   // UNI[2929] := 16#94A6;
   // UNI[2930] := 16#4FB5;
   // UNI[2931] := 16#4EB2;
   // UNI[2932] := 16#79E6;
   // UNI[2933] := 16#7434;
   // UNI[2934] := 16#52E4;
   // UNI[2935] := 16#82B9;
   // UNI[2936] := 16#64D2;
   // UNI[2937] := 16#79BD;
   // UNI[2938] := 16#5BDD;
   // UNI[2939] := 16#6C81;
   // UNI[2940] := 16#9752;
   // UNI[2941] := 16#8F7B;
   // UNI[2942] := 16#6C22;
   // UNI[2943] := 16#503E;
   // UNI[2944] := 16#537F;
   // UNI[2945] := 16#6E05;
   // UNI[2946] := 16#64CE;
   // UNI[2947] := 16#6674;
   // UNI[2948] := 16#6C30;
   // UNI[2949] := 16#60C5;
   // UNI[2950] := 16#9877;
   // UNI[2951] := 16#8BF7;
   // UNI[2952] := 16#5E86;
   // UNI[2953] := 16#743C;
   // UNI[2954] := 16#7A77;
   // UNI[2955] := 16#79CB;
   // UNI[2956] := 16#4E18;
   // UNI[2957] := 16#90B1;
   // UNI[2958] := 16#7403;
   // UNI[2959] := 16#6C42;
   // UNI[2960] := 16#56DA;
   // UNI[2961] := 16#914B;
   // UNI[2962] := 16#6CC5;
   // UNI[2963] := 16#8D8B;
   // UNI[2964] := 16#533A;
   // UNI[2965] := 16#86C6;
   // UNI[2966] := 16#66F2;
   // UNI[2967] := 16#8EAF;
   // UNI[2968] := 16#5C48;
   // UNI[2969] := 16#9A71;
   // UNI[2970] := 16#6E20;
   // UNI[2971] := 16#53D6;
   // UNI[2972] := 16#5A36;
   // UNI[2973] := 16#9F8B;
   // UNI[2974] := 16#8DA3;
   // UNI[2975] := 16#53BB;
   // UNI[2976] := 16#5708;
   // UNI[2977] := 16#98A7;
   // UNI[2978] := 16#6743;
   // UNI[2979] := 16#919B;
   // UNI[2980] := 16#6CC9;
   // UNI[2981] := 16#5168;
   // UNI[2982] := 16#75CA;
   // UNI[2983] := 16#62F3;
   // UNI[2984] := 16#72AC;
   // UNI[2985] := 16#5238;
   // UNI[2986] := 16#529D;
   // UNI[2987] := 16#7F3A;
   // UNI[2988] := 16#7094;
   // UNI[2989] := 16#7638;
   // UNI[2990] := 16#5374;
   // UNI[2991] := 16#9E4A;
   // UNI[2992] := 16#69B7;
   // UNI[2993] := 16#786E;
   // UNI[2994] := 16#96C0;
   // UNI[2995] := 16#88D9;
   // UNI[2996] := 16#7FA4;
   // UNI[2997] := 16#7136;
   // UNI[2998] := 16#71C3;
   // UNI[2999] := 16#5189;
   // UNI[3000] := 16#67D3;
   // UNI[3001] := 16#74E4;
   // UNI[3002] := 16#58E4;
   // UNI[3003] := 16#6518;
   // UNI[3004] := 16#56B7;
   // UNI[3005] := 16#8BA9;
   // UNI[3006] := 16#9976;
   // UNI[3007] := 16#6270;
   // UNI[3008] := 16#7ED5;
   // UNI[3009] := 16#60F9;
   // UNI[3010] := 16#70ED;
   // UNI[3011] := 16#58EC;
   // UNI[3012] := 16#4EC1;
   // UNI[3013] := 16#4EBA;
   // UNI[3014] := 16#5FCD;
   // UNI[3015] := 16#97E7;
   // UNI[3016] := 16#4EFB;
   // UNI[3017] := 16#8BA4;
   // UNI[3018] := 16#5203;
   // UNI[3019] := 16#598A;
   // UNI[3020] := 16#7EAB;
   // UNI[3021] := 16#6254;
   // UNI[3022] := 16#4ECD;
   // UNI[3023] := 16#65E5;
   // UNI[3024] := 16#620E;
   // UNI[3025] := 16#8338;
   // UNI[3026] := 16#84C9;
   // UNI[3027] := 16#8363;
   // UNI[3028] := 16#878D;
   // UNI[3029] := 16#7194;
   // UNI[3030] := 16#6EB6;
   // UNI[3031] := 16#5BB9;
   // UNI[3032] := 16#7ED2;
   // UNI[3033] := 16#5197;
   // UNI[3034] := 16#63C9;
   // UNI[3035] := 16#67D4;
   // UNI[3036] := 16#8089;
   // UNI[3037] := 16#8339;
   // UNI[3038] := 16#8815;
   // UNI[3039] := 16#5112;
   // UNI[3040] := 16#5B7A;
   // UNI[3041] := 16#5982;
   // UNI[3042] := 16#8FB1;
   // UNI[3043] := 16#4E73;
   // UNI[3044] := 16#6C5D;
   // UNI[3045] := 16#5165;
   // UNI[3046] := 16#8925;
   // UNI[3047] := 16#8F6F;
   // UNI[3048] := 16#962E;
   // UNI[3049] := 16#854A;
   // UNI[3050] := 16#745E;
   // UNI[3051] := 16#9510;
   // UNI[3052] := 16#95F0;
   // UNI[3053] := 16#6DA6;
   // UNI[3054] := 16#82E5;
   // UNI[3055] := 16#5F31;
   // UNI[3056] := 16#6492;
   // UNI[3057] := 16#6D12;
   // UNI[3058] := 16#8428;
   // UNI[3059] := 16#816E;
   // UNI[3060] := 16#9CC3;
   // UNI[3061] := 16#585E;
   // UNI[3062] := 16#8D5B;
   // UNI[3063] := 16#4E09;
   // UNI[3064] := 16#53C1;
   // UNI[3065] := 16#4F1E;
   // UNI[3066] := 16#6563;
   // UNI[3067] := 16#6851;
   // UNI[3068] := 16#55D3;
   // UNI[3069] := 16#4E27;
   // UNI[3070] := 16#6414;
   // UNI[3071] := 16#9A9A;
   // UNI[3072] := 16#626B;
   // UNI[3073] := 16#5AC2;
   // UNI[3074] := 16#745F;
   // UNI[3075] := 16#8272;
   // UNI[3076] := 16#6DA9;
   // UNI[3077] := 16#68EE;
   // UNI[3078] := 16#50E7;
   // UNI[3079] := 16#838E;
   // UNI[3080] := 16#7802;
   // UNI[3081] := 16#6740;
   // UNI[3082] := 16#5239;
   // UNI[3083] := 16#6C99;
   // UNI[3084] := 16#7EB1;
   // UNI[3085] := 16#50BB;
   // UNI[3086] := 16#5565;
   // UNI[3087] := 16#715E;
   // UNI[3088] := 16#7B5B;
   // UNI[3089] := 16#6652;
   // UNI[3090] := 16#73CA;
   // UNI[3091] := 16#82EB;
   // UNI[3092] := 16#6749;
   // UNI[3093] := 16#5C71;
   // UNI[3094] := 16#5220;
   // UNI[3095] := 16#717D;
   // UNI[3096] := 16#886B;
   // UNI[3097] := 16#95EA;
   // UNI[3098] := 16#9655;
   // UNI[3099] := 16#64C5;
   // UNI[3100] := 16#8D61;
   // UNI[3101] := 16#81B3;
   // UNI[3102] := 16#5584;
   // UNI[3103] := 16#6C55;
   // UNI[3104] := 16#6247;
   // UNI[3105] := 16#7F2E;
   // UNI[3106] := 16#5892;
   // UNI[3107] := 16#4F24;
   // UNI[3108] := 16#5546;
   // UNI[3109] := 16#8D4F;
   // UNI[3110] := 16#664C;
   // UNI[3111] := 16#4E0A;
   // UNI[3112] := 16#5C1A;
   // UNI[3113] := 16#88F3;
   // UNI[3114] := 16#68A2;
   // UNI[3115] := 16#634E;
   // UNI[3116] := 16#7A0D;
   // UNI[3117] := 16#70E7;
   // UNI[3118] := 16#828D;
   // UNI[3119] := 16#52FA;
   // UNI[3120] := 16#97F6;
   // UNI[3121] := 16#5C11;
   // UNI[3122] := 16#54E8;
   // UNI[3123] := 16#90B5;
   // UNI[3124] := 16#7ECD;
   // UNI[3125] := 16#5962;
   // UNI[3126] := 16#8D4A;
   // UNI[3127] := 16#86C7;
   // UNI[3128] := 16#820C;
   // UNI[3129] := 16#820D;
   // UNI[3130] := 16#8D66;
   // UNI[3131] := 16#6444;
   // UNI[3132] := 16#5C04;
   // UNI[3133] := 16#6151;
   // UNI[3134] := 16#6D89;
   // UNI[3135] := 16#793E;
   // UNI[3136] := 16#8BBE;
   // UNI[3137] := 16#7837;
   // UNI[3138] := 16#7533;
   // UNI[3139] := 16#547B;
   // UNI[3140] := 16#4F38;
   // UNI[3141] := 16#8EAB;
   // UNI[3142] := 16#6DF1;
   // UNI[3143] := 16#5A20;
   // UNI[3144] := 16#7EC5;
   // UNI[3145] := 16#795E;
   // UNI[3146] := 16#6C88;
   // UNI[3147] := 16#5BA1;
   // UNI[3148] := 16#5A76;
   // UNI[3149] := 16#751A;
   // UNI[3150] := 16#80BE;
   // UNI[3151] := 16#614E;
   // UNI[3152] := 16#6E17;
   // UNI[3153] := 16#58F0;
   // UNI[3154] := 16#751F;
   // UNI[3155] := 16#7525;
   // UNI[3156] := 16#7272;
   // UNI[3157] := 16#5347;
   // UNI[3158] := 16#7EF3;
   // UNI[3159] := 16#7701;
   // UNI[3160] := 16#76DB;
   // UNI[3161] := 16#5269;
   // UNI[3162] := 16#80DC;
   // UNI[3163] := 16#5723;
   // UNI[3164] := 16#5E08;
   // UNI[3165] := 16#5931;
   // UNI[3166] := 16#72EE;
   // UNI[3167] := 16#65BD;
   // UNI[3168] := 16#6E7F;
   // UNI[3169] := 16#8BD7;
   // UNI[3170] := 16#5C38;
   // UNI[3171] := 16#8671;
   // UNI[3172] := 16#5341;
   // UNI[3173] := 16#77F3;
   // UNI[3174] := 16#62FE;
   // UNI[3175] := 16#65F6;
   // UNI[3176] := 16#4EC0;
   // UNI[3177] := 16#98DF;
   // UNI[3178] := 16#8680;
   // UNI[3179] := 16#5B9E;
   // UNI[3180] := 16#8BC6;
   // UNI[3181] := 16#53F2;
   // UNI[3182] := 16#77E2;
   // UNI[3183] := 16#4F7F;
   // UNI[3184] := 16#5C4E;
   // UNI[3185] := 16#9A76;
   // UNI[3186] := 16#59CB;
   // UNI[3187] := 16#5F0F;
   // UNI[3188] := 16#793A;
   // UNI[3189] := 16#58EB;
   // UNI[3190] := 16#4E16;
   // UNI[3191] := 16#67FF;
   // UNI[3192] := 16#4E8B;
   // UNI[3193] := 16#62ED;
   // UNI[3194] := 16#8A93;
   // UNI[3195] := 16#901D;
   // UNI[3196] := 16#52BF;
   // UNI[3197] := 16#662F;
   // UNI[3198] := 16#55DC;
   // UNI[3199] := 16#566C;
   // UNI[3200] := 16#9002;
   // UNI[3201] := 16#4ED5;
   // UNI[3202] := 16#4F8D;
   // UNI[3203] := 16#91CA;
   // UNI[3204] := 16#9970;
   // UNI[3205] := 16#6C0F;
   // UNI[3206] := 16#5E02;
   // UNI[3207] := 16#6043;
   // UNI[3208] := 16#5BA4;
   // UNI[3209] := 16#89C6;
   // UNI[3210] := 16#8BD5;
   // UNI[3211] := 16#6536;
   // UNI[3212] := 16#624B;
   // UNI[3213] := 16#9996;
   // UNI[3214] := 16#5B88;
   // UNI[3215] := 16#5BFF;
   // UNI[3216] := 16#6388;
   // UNI[3217] := 16#552E;
   // UNI[3218] := 16#53D7;
   // UNI[3219] := 16#7626;
   // UNI[3220] := 16#517D;
   // UNI[3221] := 16#852C;
   // UNI[3222] := 16#67A2;
   // UNI[3223] := 16#68B3;
   // UNI[3224] := 16#6B8A;
   // UNI[3225] := 16#6292;
   // UNI[3226] := 16#8F93;
   // UNI[3227] := 16#53D4;
   // UNI[3228] := 16#8212;
   // UNI[3229] := 16#6DD1;
   // UNI[3230] := 16#758F;
   // UNI[3231] := 16#4E66;
   // UNI[3232] := 16#8D4E;
   // UNI[3233] := 16#5B70;
   // UNI[3234] := 16#719F;
   // UNI[3235] := 16#85AF;
   // UNI[3236] := 16#6691;
   // UNI[3237] := 16#66D9;
   // UNI[3238] := 16#7F72;
   // UNI[3239] := 16#8700;
   // UNI[3240] := 16#9ECD;
   // UNI[3241] := 16#9F20;
   // UNI[3242] := 16#5C5E;
   // UNI[3243] := 16#672F;
   // UNI[3244] := 16#8FF0;
   // UNI[3245] := 16#6811;
   // UNI[3246] := 16#675F;
   // UNI[3247] := 16#620D;
   // UNI[3248] := 16#7AD6;
   // UNI[3249] := 16#5885;
   // UNI[3250] := 16#5EB6;
   // UNI[3251] := 16#6570;
   // UNI[3252] := 16#6F31;
   // UNI[3253] := 16#6055;
   // UNI[3254] := 16#5237;
   // UNI[3255] := 16#800D;
   // UNI[3256] := 16#6454;
   // UNI[3257] := 16#8870;
   // UNI[3258] := 16#7529;
   // UNI[3259] := 16#5E05;
   // UNI[3260] := 16#6813;
   // UNI[3261] := 16#62F4;
   // UNI[3262] := 16#971C;
   // UNI[3263] := 16#53CC;
   // UNI[3264] := 16#723D;
   // UNI[3265] := 16#8C01;
   // UNI[3266] := 16#6C34;
   // UNI[3267] := 16#7761;
   // UNI[3268] := 16#7A0E;
   // UNI[3269] := 16#542E;
   // UNI[3270] := 16#77AC;
   // UNI[3271] := 16#987A;
   // UNI[3272] := 16#821C;
   // UNI[3273] := 16#8BF4;
   // UNI[3274] := 16#7855;
   // UNI[3275] := 16#6714;
   // UNI[3276] := 16#70C1;
   // UNI[3277] := 16#65AF;
   // UNI[3278] := 16#6495;
   // UNI[3279] := 16#5636;
   // UNI[3280] := 16#601D;
   // UNI[3281] := 16#79C1;
   // UNI[3282] := 16#53F8;
   // UNI[3283] := 16#4E1D;
   // UNI[3284] := 16#6B7B;
   // UNI[3285] := 16#8086;
   // UNI[3286] := 16#5BFA;
   // UNI[3287] := 16#55E3;
   // UNI[3288] := 16#56DB;
   // UNI[3289] := 16#4F3A;
   // UNI[3290] := 16#4F3C;
   // UNI[3291] := 16#9972;
   // UNI[3292] := 16#5DF3;
   // UNI[3293] := 16#677E;
   // UNI[3294] := 16#8038;
   // UNI[3295] := 16#6002;
   // UNI[3296] := 16#9882;
   // UNI[3297] := 16#9001;
   // UNI[3298] := 16#5B8B;
   // UNI[3299] := 16#8BBC;
   // UNI[3300] := 16#8BF5;
   // UNI[3301] := 16#641C;
   // UNI[3302] := 16#8258;
   // UNI[3303] := 16#64DE;
   // UNI[3304] := 16#55FD;
   // UNI[3305] := 16#82CF;
   // UNI[3306] := 16#9165;
   // UNI[3307] := 16#4FD7;
   // UNI[3308] := 16#7D20;
   // UNI[3309] := 16#901F;
   // UNI[3310] := 16#7C9F;
   // UNI[3311] := 16#50F3;
   // UNI[3312] := 16#5851;
   // UNI[3313] := 16#6EAF;
   // UNI[3314] := 16#5BBF;
   // UNI[3315] := 16#8BC9;
   // UNI[3316] := 16#8083;
   // UNI[3317] := 16#9178;
   // UNI[3318] := 16#849C;
   // UNI[3319] := 16#7B97;
   // UNI[3320] := 16#867D;
   // UNI[3321] := 16#968B;
   // UNI[3322] := 16#968F;
   // UNI[3323] := 16#7EE5;
   // UNI[3324] := 16#9AD3;
   // UNI[3325] := 16#788E;
   // UNI[3326] := 16#5C81;
   // UNI[3327] := 16#7A57;
   // UNI[3328] := 16#9042;
   // UNI[3329] := 16#96A7;
   // UNI[3330] := 16#795F;
   // UNI[3331] := 16#5B59;
   // UNI[3332] := 16#635F;
   // UNI[3333] := 16#7B0B;
   // UNI[3334] := 16#84D1;
   // UNI[3335] := 16#68AD;
   // UNI[3336] := 16#5506;
   // UNI[3337] := 16#7F29;
   // UNI[3338] := 16#7410;
   // UNI[3339] := 16#7D22;
   // UNI[3340] := 16#9501;
   // UNI[3341] := 16#6240;
   // UNI[3342] := 16#584C;
   // UNI[3343] := 16#4ED6;
   // UNI[3344] := 16#5B83;
   // UNI[3345] := 16#5979;
   // UNI[3346] := 16#5854;
   // UNI[3347] := 16#736D;
   // UNI[3348] := 16#631E;
   // UNI[3349] := 16#8E4B;
   // UNI[3350] := 16#8E0F;
   // UNI[3351] := 16#80CE;
   // UNI[3352] := 16#82D4;
   // UNI[3353] := 16#62AC;
   // UNI[3354] := 16#53F0;
   // UNI[3355] := 16#6CF0;
   // UNI[3356] := 16#915E;
   // UNI[3357] := 16#592A;
   // UNI[3358] := 16#6001;
   // UNI[3359] := 16#6C70;
   // UNI[3360] := 16#574D;
   // UNI[3361] := 16#644A;
   // UNI[3362] := 16#8D2A;
   // UNI[3363] := 16#762B;
   // UNI[3364] := 16#6EE9;
   // UNI[3365] := 16#575B;
   // UNI[3366] := 16#6A80;
   // UNI[3367] := 16#75F0;
   // UNI[3368] := 16#6F6D;
   // UNI[3369] := 16#8C2D;
   // UNI[3370] := 16#8C08;
   // UNI[3371] := 16#5766;
   // UNI[3372] := 16#6BEF;
   // UNI[3373] := 16#8892;
   // UNI[3374] := 16#78B3;
   // UNI[3375] := 16#63A2;
   // UNI[3376] := 16#53F9;
   // UNI[3377] := 16#70AD;
   // UNI[3378] := 16#6C64;
   // UNI[3379] := 16#5858;
   // UNI[3380] := 16#642A;
   // UNI[3381] := 16#5802;
   // UNI[3382] := 16#68E0;
   // UNI[3383] := 16#819B;
   // UNI[3384] := 16#5510;
   // UNI[3385] := 16#7CD6;
   // UNI[3386] := 16#5018;
   // UNI[3387] := 16#8EBA;
   // UNI[3388] := 16#6DCC;
   // UNI[3389] := 16#8D9F;
   // UNI[3390] := 16#70EB;
   // UNI[3391] := 16#638F;
   // UNI[3392] := 16#6D9B;
   // UNI[3393] := 16#6ED4;
   // UNI[3394] := 16#7EE6;
   // UNI[3395] := 16#8404;
   // UNI[3396] := 16#6843;
   // UNI[3397] := 16#9003;
   // UNI[3398] := 16#6DD8;
   // UNI[3399] := 16#9676;
   // UNI[3400] := 16#8BA8;
   // UNI[3401] := 16#5957;
   // UNI[3402] := 16#7279;
   // UNI[3403] := 16#85E4;
   // UNI[3404] := 16#817E;
   // UNI[3405] := 16#75BC;
   // UNI[3406] := 16#8A8A;
   // UNI[3407] := 16#68AF;
   // UNI[3408] := 16#5254;
   // UNI[3409] := 16#8E22;
   // UNI[3410] := 16#9511;
   // UNI[3411] := 16#63D0;
   // UNI[3412] := 16#9898;
   // UNI[3413] := 16#8E44;
   // UNI[3414] := 16#557C;
   // UNI[3415] := 16#4F53;
   // UNI[3416] := 16#66FF;
   // UNI[3417] := 16#568F;
   // UNI[3418] := 16#60D5;
   // UNI[3419] := 16#6D95;
   // UNI[3420] := 16#5243;
   // UNI[3421] := 16#5C49;
   // UNI[3422] := 16#5929;
   // UNI[3423] := 16#6DFB;
   // UNI[3424] := 16#586B;
   // UNI[3425] := 16#7530;
   // UNI[3426] := 16#751C;
   // UNI[3427] := 16#606C;
   // UNI[3428] := 16#8214;
   // UNI[3429] := 16#8146;
   // UNI[3430] := 16#6311;
   // UNI[3431] := 16#6761;
   // UNI[3432] := 16#8FE2;
   // UNI[3433] := 16#773A;
   // UNI[3434] := 16#8DF3;
   // UNI[3435] := 16#8D34;
   // UNI[3436] := 16#94C1;
   // UNI[3437] := 16#5E16;
   // UNI[3438] := 16#5385;
   // UNI[3439] := 16#542C;
   // UNI[3440] := 16#70C3;
   // UNI[3441] := 16#6C40;
   // UNI[3442] := 16#5EF7;
   // UNI[3443] := 16#505C;
   // UNI[3444] := 16#4EAD;
   // UNI[3445] := 16#5EAD;
   // UNI[3446] := 16#633A;
   // UNI[3447] := 16#8247;
   // UNI[3448] := 16#901A;
   // UNI[3449] := 16#6850;
   // UNI[3450] := 16#916E;
   // UNI[3451] := 16#77B3;
   // UNI[3452] := 16#540C;
   // UNI[3453] := 16#94DC;
   // UNI[3454] := 16#5F64;
   // UNI[3455] := 16#7AE5;
   // UNI[3456] := 16#6876;
   // UNI[3457] := 16#6345;
   // UNI[3458] := 16#7B52;
   // UNI[3459] := 16#7EDF;
   // UNI[3460] := 16#75DB;
   // UNI[3461] := 16#5077;
   // UNI[3462] := 16#6295;
   // UNI[3463] := 16#5934;
   // UNI[3464] := 16#900F;
   // UNI[3465] := 16#51F8;
   // UNI[3466] := 16#79C3;
   // UNI[3467] := 16#7A81;
   // UNI[3468] := 16#56FE;
   // UNI[3469] := 16#5F92;
   // UNI[3470] := 16#9014;
   // UNI[3471] := 16#6D82;
   // UNI[3472] := 16#5C60;
   // UNI[3473] := 16#571F;
   // UNI[3474] := 16#5410;
   // UNI[3475] := 16#5154;
   // UNI[3476] := 16#6E4D;
   // UNI[3477] := 16#56E2;
   // UNI[3478] := 16#63A8;
   // UNI[3479] := 16#9893;
   // UNI[3480] := 16#817F;
   // UNI[3481] := 16#8715;
   // UNI[3482] := 16#892A;
   // UNI[3483] := 16#9000;
   // UNI[3484] := 16#541E;
   // UNI[3485] := 16#5C6F;
   // UNI[3486] := 16#81C0;
   // UNI[3487] := 16#62D6;
   // UNI[3488] := 16#6258;
   // UNI[3489] := 16#8131;
   // UNI[3490] := 16#9E35;
   // UNI[3491] := 16#9640;
   // UNI[3492] := 16#9A6E;
   // UNI[3493] := 16#9A7C;
   // UNI[3494] := 16#692D;
   // UNI[3495] := 16#59A5;
   // UNI[3496] := 16#62D3;
   // UNI[3497] := 16#553E;
   // UNI[3498] := 16#6316;
   // UNI[3499] := 16#54C7;
   // UNI[3500] := 16#86D9;
   // UNI[3501] := 16#6D3C;
   // UNI[3502] := 16#5A03;
   // UNI[3503] := 16#74E6;
   // UNI[3504] := 16#889C;
   // UNI[3505] := 16#6B6A;
   // UNI[3506] := 16#5916;
   // UNI[3507] := 16#8C4C;
   // UNI[3508] := 16#5F2F;
   // UNI[3509] := 16#6E7E;
   // UNI[3510] := 16#73A9;
   // UNI[3511] := 16#987D;
   // UNI[3512] := 16#4E38;
   // UNI[3513] := 16#70F7;
   // UNI[3514] := 16#5B8C;
   // UNI[3515] := 16#7897;
   // UNI[3516] := 16#633D;
   // UNI[3517] := 16#665A;
   // UNI[3518] := 16#7696;
   // UNI[3519] := 16#60CB;
   // UNI[3520] := 16#5B9B;
   // UNI[3521] := 16#5A49;
   // UNI[3522] := 16#4E07;
   // UNI[3523] := 16#8155;
   // UNI[3524] := 16#6C6A;
   // UNI[3525] := 16#738B;
   // UNI[3526] := 16#4EA1;
   // UNI[3527] := 16#6789;
   // UNI[3528] := 16#7F51;
   // UNI[3529] := 16#5F80;
   // UNI[3530] := 16#65FA;
   // UNI[3531] := 16#671B;
   // UNI[3532] := 16#5FD8;
   // UNI[3533] := 16#5984;
   // UNI[3534] := 16#5A01;
   // UNI[3535] := 16#5DCD;
   // UNI[3536] := 16#5FAE;
   // UNI[3537] := 16#5371;
   // UNI[3538] := 16#97E6;
   // UNI[3539] := 16#8FDD;
   // UNI[3540] := 16#6845;
   // UNI[3541] := 16#56F4;
   // UNI[3542] := 16#552F;
   // UNI[3543] := 16#60DF;
   // UNI[3544] := 16#4E3A;
   // UNI[3545] := 16#6F4D;
   // UNI[3546] := 16#7EF4;
   // UNI[3547] := 16#82C7;
   // UNI[3548] := 16#840E;
   // UNI[3549] := 16#59D4;
   // UNI[3550] := 16#4F1F;
   // UNI[3551] := 16#4F2A;
   // UNI[3552] := 16#5C3E;
   // UNI[3553] := 16#7EAC;
   // UNI[3554] := 16#672A;
   // UNI[3555] := 16#851A;
   // UNI[3556] := 16#5473;
   // UNI[3557] := 16#754F;
   // UNI[3558] := 16#80C3;
   // UNI[3559] := 16#5582;
   // UNI[3560] := 16#9B4F;
   // UNI[3561] := 16#4F4D;
   // UNI[3562] := 16#6E2D;
   // UNI[3563] := 16#8C13;
   // UNI[3564] := 16#5C09;
   // UNI[3565] := 16#6170;
   // UNI[3566] := 16#536B;
   // UNI[3567] := 16#761F;
   // UNI[3568] := 16#6E29;
   // UNI[3569] := 16#868A;
   // UNI[3570] := 16#6587;
   // UNI[3571] := 16#95FB;
   // UNI[3572] := 16#7EB9;
   // UNI[3573] := 16#543B;
   // UNI[3574] := 16#7A33;
   // UNI[3575] := 16#7D0A;
   // UNI[3576] := 16#95EE;
   // UNI[3577] := 16#55E1;
   // UNI[3578] := 16#7FC1;
   // UNI[3579] := 16#74EE;
   // UNI[3580] := 16#631D;
   // UNI[3581] := 16#8717;
   // UNI[3582] := 16#6DA1;
   // UNI[3583] := 16#7A9D;
   // UNI[3584] := 16#6211;
   // UNI[3585] := 16#65A1;
   // UNI[3586] := 16#5367;
   // UNI[3587] := 16#63E1;
   // UNI[3588] := 16#6C83;
   // UNI[3589] := 16#5DEB;
   // UNI[3590] := 16#545C;
   // UNI[3591] := 16#94A8;
   // UNI[3592] := 16#4E4C;
   // UNI[3593] := 16#6C61;
   // UNI[3594] := 16#8BEC;
   // UNI[3595] := 16#5C4B;
   // UNI[3596] := 16#65E0;
   // UNI[3597] := 16#829C;
   // UNI[3598] := 16#68A7;
   // UNI[3599] := 16#543E;
   // UNI[3600] := 16#5434;
   // UNI[3601] := 16#6BCB;
   // UNI[3602] := 16#6B66;
   // UNI[3603] := 16#4E94;
   // UNI[3604] := 16#6342;
   // UNI[3605] := 16#5348;
   // UNI[3606] := 16#821E;
   // UNI[3607] := 16#4F0D;
   // UNI[3608] := 16#4FAE;
   // UNI[3609] := 16#575E;
   // UNI[3610] := 16#620A;
   // UNI[3611] := 16#96FE;
   // UNI[3612] := 16#6664;
   // UNI[3613] := 16#7269;
   // UNI[3614] := 16#52FF;
   // UNI[3615] := 16#52A1;
   // UNI[3616] := 16#609F;
   // UNI[3617] := 16#8BEF;
   // UNI[3618] := 16#6614;
   // UNI[3619] := 16#7199;
   // UNI[3620] := 16#6790;
   // UNI[3621] := 16#897F;
   // UNI[3622] := 16#7852;
   // UNI[3623] := 16#77FD;
   // UNI[3624] := 16#6670;
   // UNI[3625] := 16#563B;
   // UNI[3626] := 16#5438;
   // UNI[3627] := 16#9521;
   // UNI[3628] := 16#727A;
   // UNI[3629] := 16#7A00;
   // UNI[3630] := 16#606F;
   // UNI[3631] := 16#5E0C;
   // UNI[3632] := 16#6089;
   // UNI[3633] := 16#819D;
   // UNI[3634] := 16#5915;
   // UNI[3635] := 16#60DC;
   // UNI[3636] := 16#7184;
   // UNI[3637] := 16#70EF;
   // UNI[3638] := 16#6EAA;
   // UNI[3639] := 16#6C50;
   // UNI[3640] := 16#7280;
   // UNI[3641] := 16#6A84;
   // UNI[3642] := 16#88AD;
   // UNI[3643] := 16#5E2D;
   // UNI[3644] := 16#4E60;
   // UNI[3645] := 16#5AB3;
   // UNI[3646] := 16#559C;
   // UNI[3647] := 16#94E3;
   // UNI[3648] := 16#6D17;
   // UNI[3649] := 16#7CFB;
   // UNI[3650] := 16#9699;
   // UNI[3651] := 16#620F;
   // UNI[3652] := 16#7EC6;
   // UNI[3653] := 16#778E;
   // UNI[3654] := 16#867E;
   // UNI[3655] := 16#5323;
   // UNI[3656] := 16#971E;
   // UNI[3657] := 16#8F96;
   // UNI[3658] := 16#6687;
   // UNI[3659] := 16#5CE1;
   // UNI[3660] := 16#4FA0;
   // UNI[3661] := 16#72ED;
   // UNI[3662] := 16#4E0B;
   // UNI[3663] := 16#53A6;
   // UNI[3664] := 16#590F;
   // UNI[3665] := 16#5413;
   // UNI[3666] := 16#6380;
   // UNI[3667] := 16#9528;
   // UNI[3668] := 16#5148;
   // UNI[3669] := 16#4ED9;
   // UNI[3670] := 16#9C9C;
   // UNI[3671] := 16#7EA4;
   // UNI[3672] := 16#54B8;
   // UNI[3673] := 16#8D24;
   // UNI[3674] := 16#8854;
   // UNI[3675] := 16#8237;
   // UNI[3676] := 16#95F2;
   // UNI[3677] := 16#6D8E;
   // UNI[3678] := 16#5F26;
   // UNI[3679] := 16#5ACC;
   // UNI[3680] := 16#663E;
   // UNI[3681] := 16#9669;
   // UNI[3682] := 16#73B0;
   // UNI[3683] := 16#732E;
   // UNI[3684] := 16#53BF;
   // UNI[3685] := 16#817A;
   // UNI[3686] := 16#9985;
   // UNI[3687] := 16#7FA1;
   // UNI[3688] := 16#5BAA;
   // UNI[3689] := 16#9677;
   // UNI[3690] := 16#9650;
   // UNI[3691] := 16#7EBF;
   // UNI[3692] := 16#76F8;
   // UNI[3693] := 16#53A2;
   // UNI[3694] := 16#9576;
   // UNI[3695] := 16#9999;
   // UNI[3696] := 16#7BB1;
   // UNI[3697] := 16#8944;
   // UNI[3698] := 16#6E58;
   // UNI[3699] := 16#4E61;
   // UNI[3700] := 16#7FD4;
   // UNI[3701] := 16#7965;
   // UNI[3702] := 16#8BE6;
   // UNI[3703] := 16#60F3;
   // UNI[3704] := 16#54CD;
   // UNI[3705] := 16#4EAB;
   // UNI[3706] := 16#9879;
   // UNI[3707] := 16#5DF7;
   // UNI[3708] := 16#6A61;
   // UNI[3709] := 16#50CF;
   // UNI[3710] := 16#5411;
   // UNI[3711] := 16#8C61;
   // UNI[3712] := 16#8427;
   // UNI[3713] := 16#785D;
   // UNI[3714] := 16#9704;
   // UNI[3715] := 16#524A;
   // UNI[3716] := 16#54EE;
   // UNI[3717] := 16#56A3;
   // UNI[3718] := 16#9500;
   // UNI[3719] := 16#6D88;
   // UNI[3720] := 16#5BB5;
   // UNI[3721] := 16#6DC6;
   // UNI[3722] := 16#6653;
   // UNI[3723] := 16#5C0F;
   // UNI[3724] := 16#5B5D;
   // UNI[3725] := 16#6821;
   // UNI[3726] := 16#8096;
   // UNI[3727] := 16#5578;
   // UNI[3728] := 16#7B11;
   // UNI[3729] := 16#6548;
   // UNI[3730] := 16#6954;
   // UNI[3731] := 16#4E9B;
   // UNI[3732] := 16#6B47;
   // UNI[3733] := 16#874E;
   // UNI[3734] := 16#978B;
   // UNI[3735] := 16#534F;
   // UNI[3736] := 16#631F;
   // UNI[3737] := 16#643A;
   // UNI[3738] := 16#90AA;
   // UNI[3739] := 16#659C;
   // UNI[3740] := 16#80C1;
   // UNI[3741] := 16#8C10;
   // UNI[3742] := 16#5199;
   // UNI[3743] := 16#68B0;
   // UNI[3744] := 16#5378;
   // UNI[3745] := 16#87F9;
   // UNI[3746] := 16#61C8;
   // UNI[3747] := 16#6CC4;
   // UNI[3748] := 16#6CFB;
   // UNI[3749] := 16#8C22;
   // UNI[3750] := 16#5C51;
   // UNI[3751] := 16#85AA;
   // UNI[3752] := 16#82AF;
   // UNI[3753] := 16#950C;
   // UNI[3754] := 16#6B23;
   // UNI[3755] := 16#8F9B;
   // UNI[3756] := 16#65B0;
   // UNI[3757] := 16#5FFB;
   // UNI[3758] := 16#5FC3;
   // UNI[3759] := 16#4FE1;
   // UNI[3760] := 16#8845;
   // UNI[3761] := 16#661F;
   // UNI[3762] := 16#8165;
   // UNI[3763] := 16#7329;
   // UNI[3764] := 16#60FA;
   // UNI[3765] := 16#5174;
   // UNI[3766] := 16#5211;
   // UNI[3767] := 16#578B;
   // UNI[3768] := 16#5F62;
   // UNI[3769] := 16#90A2;
   // UNI[3770] := 16#884C;
   // UNI[3771] := 16#9192;
   // UNI[3772] := 16#5E78;
   // UNI[3773] := 16#674F;
   // UNI[3774] := 16#6027;
   // UNI[3775] := 16#59D3;
   // UNI[3776] := 16#5144;
   // UNI[3777] := 16#51F6;
   // UNI[3778] := 16#80F8;
   // UNI[3779] := 16#5308;
   // UNI[3780] := 16#6C79;
   // UNI[3781] := 16#96C4;
   // UNI[3782] := 16#718A;
   // UNI[3783] := 16#4F11;
   // UNI[3784] := 16#4FEE;
   // UNI[3785] := 16#7F9E;
   // UNI[3786] := 16#673D;
   // UNI[3787] := 16#55C5;
   // UNI[3788] := 16#9508;
   // UNI[3789] := 16#79C0;
   // UNI[3790] := 16#8896;
   // UNI[3791] := 16#7EE3;
   // UNI[3792] := 16#589F;
   // UNI[3793] := 16#620C;
   // UNI[3794] := 16#9700;
   // UNI[3795] := 16#865A;
   // UNI[3796] := 16#5618;
   // UNI[3797] := 16#987B;
   // UNI[3798] := 16#5F90;
   // UNI[3799] := 16#8BB8;
   // UNI[3800] := 16#84C4;
   // UNI[3801] := 16#9157;
   // UNI[3802] := 16#53D9;
   // UNI[3803] := 16#65ED;
   // UNI[3804] := 16#5E8F;
   // UNI[3805] := 16#755C;
   // UNI[3806] := 16#6064;
   // UNI[3807] := 16#7D6E;
   // UNI[3808] := 16#5A7F;
   // UNI[3809] := 16#7EEA;
   // UNI[3810] := 16#7EED;
   // UNI[3811] := 16#8F69;
   // UNI[3812] := 16#55A7;
   // UNI[3813] := 16#5BA3;
   // UNI[3814] := 16#60AC;
   // UNI[3815] := 16#65CB;
   // UNI[3816] := 16#7384;
   // UNI[3817] := 16#9009;
   // UNI[3818] := 16#7663;
   // UNI[3819] := 16#7729;
   // UNI[3820] := 16#7EDA;
   // UNI[3821] := 16#9774;
   // UNI[3822] := 16#859B;
   // UNI[3823] := 16#5B66;
   // UNI[3824] := 16#7A74;
   // UNI[3825] := 16#96EA;
   // UNI[3826] := 16#8840;
   // UNI[3827] := 16#52CB;
   // UNI[3828] := 16#718F;
   // UNI[3829] := 16#5FAA;
   // UNI[3830] := 16#65EC;
   // UNI[3831] := 16#8BE2;
   // UNI[3832] := 16#5BFB;
   // UNI[3833] := 16#9A6F;
   // UNI[3834] := 16#5DE1;
   // UNI[3835] := 16#6B89;
   // UNI[3836] := 16#6C5B;
   // UNI[3837] := 16#8BAD;
   // UNI[3838] := 16#8BAF;
   // UNI[3839] := 16#900A;
   // UNI[3840] := 16#8FC5;
   // UNI[3841] := 16#538B;
   // UNI[3842] := 16#62BC;
   // UNI[3843] := 16#9E26;
   // UNI[3844] := 16#9E2D;
   // UNI[3845] := 16#5440;
   // UNI[3846] := 16#4E2B;
   // UNI[3847] := 16#82BD;
   // UNI[3848] := 16#7259;
   // UNI[3849] := 16#869C;
   // UNI[3850] := 16#5D16;
   // UNI[3851] := 16#8859;
   // UNI[3852] := 16#6DAF;
   // UNI[3853] := 16#96C5;
   // UNI[3854] := 16#54D1;
   // UNI[3855] := 16#4E9A;
   // UNI[3856] := 16#8BB6;
   // UNI[3857] := 16#7109;
   // UNI[3858] := 16#54BD;
   // UNI[3859] := 16#9609;
   // UNI[3860] := 16#70DF;
   // UNI[3861] := 16#6DF9;
   // UNI[3862] := 16#76D0;
   // UNI[3863] := 16#4E25;
   // UNI[3864] := 16#7814;
   // UNI[3865] := 16#8712;
   // UNI[3866] := 16#5CA9;
   // UNI[3867] := 16#5EF6;
   // UNI[3868] := 16#8A00;
   // UNI[3869] := 16#989C;
   // UNI[3870] := 16#960E;
   // UNI[3871] := 16#708E;
   // UNI[3872] := 16#6CBF;
   // UNI[3873] := 16#5944;
   // UNI[3874] := 16#63A9;
   // UNI[3875] := 16#773C;
   // UNI[3876] := 16#884D;
   // UNI[3877] := 16#6F14;
   // UNI[3878] := 16#8273;
   // UNI[3879] := 16#5830;
   // UNI[3880] := 16#71D5;
   // UNI[3881] := 16#538C;
   // UNI[3882] := 16#781A;
   // UNI[3883] := 16#96C1;
   // UNI[3884] := 16#5501;
   // UNI[3885] := 16#5F66;
   // UNI[3886] := 16#7130;
   // UNI[3887] := 16#5BB4;
   // UNI[3888] := 16#8C1A;
   // UNI[3889] := 16#9A8C;
   // UNI[3890] := 16#6B83;
   // UNI[3891] := 16#592E;
   // UNI[3892] := 16#9E2F;
   // UNI[3893] := 16#79E7;
   // UNI[3894] := 16#6768;
   // UNI[3895] := 16#626C;
   // UNI[3896] := 16#4F6F;
   // UNI[3897] := 16#75A1;
   // UNI[3898] := 16#7F8A;
   // UNI[3899] := 16#6D0B;
   // UNI[3900] := 16#9633;
   // UNI[3901] := 16#6C27;
   // UNI[3902] := 16#4EF0;
   // UNI[3903] := 16#75D2;
   // UNI[3904] := 16#517B;
   // UNI[3905] := 16#6837;
   // UNI[3906] := 16#6F3E;
   // UNI[3907] := 16#9080;
   // UNI[3908] := 16#8170;
   // UNI[3909] := 16#5996;
   // UNI[3910] := 16#7476;
   // UNI[3911] := 16#6447;
   // UNI[3912] := 16#5C27;
   // UNI[3913] := 16#9065;
   // UNI[3914] := 16#7A91;
   // UNI[3915] := 16#8C23;
   // UNI[3916] := 16#59DA;
   // UNI[3917] := 16#54AC;
   // UNI[3918] := 16#8200;
   // UNI[3919] := 16#836F;
   // UNI[3920] := 16#8981;
   // UNI[3921] := 16#8000;
   // UNI[3922] := 16#6930;
   // UNI[3923] := 16#564E;
   // UNI[3924] := 16#8036;
   // UNI[3925] := 16#7237;
   // UNI[3926] := 16#91CE;
   // UNI[3927] := 16#51B6;
   // UNI[3928] := 16#4E5F;
   // UNI[3929] := 16#9875;
   // UNI[3930] := 16#6396;
   // UNI[3931] := 16#4E1A;
   // UNI[3932] := 16#53F6;
   // UNI[3933] := 16#66F3;
   // UNI[3934] := 16#814B;
   // UNI[3935] := 16#591C;
   // UNI[3936] := 16#6DB2;
   // UNI[3937] := 16#4E00;
   // UNI[3938] := 16#58F9;
   // UNI[3939] := 16#533B;
   // UNI[3940] := 16#63D6;
   // UNI[3941] := 16#94F1;
   // UNI[3942] := 16#4F9D;
   // UNI[3943] := 16#4F0A;
   // UNI[3944] := 16#8863;
   // UNI[3945] := 16#9890;
   // UNI[3946] := 16#5937;
   // UNI[3947] := 16#9057;
   // UNI[3948] := 16#79FB;
   // UNI[3949] := 16#4EEA;
   // UNI[3950] := 16#80F0;
   // UNI[3951] := 16#7591;
   // UNI[3952] := 16#6C82;
   // UNI[3953] := 16#5B9C;
   // UNI[3954] := 16#59E8;
   // UNI[3955] := 16#5F5D;
   // UNI[3956] := 16#6905;
   // UNI[3957] := 16#8681;
   // UNI[3958] := 16#501A;
   // UNI[3959] := 16#5DF2;
   // UNI[3960] := 16#4E59;
   // UNI[3961] := 16#77E3;
   // UNI[3962] := 16#4EE5;
   // UNI[3963] := 16#827A;
   // UNI[3964] := 16#6291;
   // UNI[3965] := 16#6613;
   // UNI[3966] := 16#9091;
   // UNI[3967] := 16#5C79;
   // UNI[3968] := 16#4EBF;
   // UNI[3969] := 16#5F79;
   // UNI[3970] := 16#81C6;
   // UNI[3971] := 16#9038;
   // UNI[3972] := 16#8084;
   // UNI[3973] := 16#75AB;
   // UNI[3974] := 16#4EA6;
   // UNI[3975] := 16#88D4;
   // UNI[3976] := 16#610F;
   // UNI[3977] := 16#6BC5;
   // UNI[3978] := 16#5FC6;
   // UNI[3979] := 16#4E49;
   // UNI[3980] := 16#76CA;
   // UNI[3981] := 16#6EA2;
   // UNI[3982] := 16#8BE3;
   // UNI[3983] := 16#8BAE;
   // UNI[3984] := 16#8C0A;
   // UNI[3985] := 16#8BD1;
   // UNI[3986] := 16#5F02;
   // UNI[3987] := 16#7FFC;
   // UNI[3988] := 16#7FCC;
   // UNI[3989] := 16#7ECE;
   // UNI[3990] := 16#8335;
   // UNI[3991] := 16#836B;
   // UNI[3992] := 16#56E0;
   // UNI[3993] := 16#6BB7;
   // UNI[3994] := 16#97F3;
   // UNI[3995] := 16#9634;
   // UNI[3996] := 16#59FB;
   // UNI[3997] := 16#541F;
   // UNI[3998] := 16#94F6;
   // UNI[3999] := 16#6DEB;
   // UNI[4000] := 16#5BC5;
   // UNI[4001] := 16#996E;
   // UNI[4002] := 16#5C39;
   // UNI[4003] := 16#5F15;
   // UNI[4004] := 16#9690;
   // UNI[4005] := 16#5370;
   // UNI[4006] := 16#82F1;
   // UNI[4007] := 16#6A31;
   // UNI[4008] := 16#5A74;
   // UNI[4009] := 16#9E70;
   // UNI[4010] := 16#5E94;
   // UNI[4011] := 16#7F28;
   // UNI[4012] := 16#83B9;
   // UNI[4013] := 16#8424;
   // UNI[4014] := 16#8425;
   // UNI[4015] := 16#8367;
   // UNI[4016] := 16#8747;
   // UNI[4017] := 16#8FCE;
   // UNI[4018] := 16#8D62;
   // UNI[4019] := 16#76C8;
   // UNI[4020] := 16#5F71;
   // UNI[4021] := 16#9896;
   // UNI[4022] := 16#786C;
   // UNI[4023] := 16#6620;
   // UNI[4024] := 16#54DF;
   // UNI[4025] := 16#62E5;
   // UNI[4026] := 16#4F63;
   // UNI[4027] := 16#81C3;
   // UNI[4028] := 16#75C8;
   // UNI[4029] := 16#5EB8;
   // UNI[4030] := 16#96CD;
   // UNI[4031] := 16#8E0A;
   // UNI[4032] := 16#86F9;
   // UNI[4033] := 16#548F;
   // UNI[4034] := 16#6CF3;
   // UNI[4035] := 16#6D8C;
   // UNI[4036] := 16#6C38;
   // UNI[4037] := 16#607F;
   // UNI[4038] := 16#52C7;
   // UNI[4039] := 16#7528;
   // UNI[4040] := 16#5E7D;
   // UNI[4041] := 16#4F18;
   // UNI[4042] := 16#60A0;
   // UNI[4043] := 16#5FE7;
   // UNI[4044] := 16#5C24;
   // UNI[4045] := 16#7531;
   // UNI[4046] := 16#90AE;
   // UNI[4047] := 16#94C0;
   // UNI[4048] := 16#72B9;
   // UNI[4049] := 16#6CB9;
   // UNI[4050] := 16#6E38;
   // UNI[4051] := 16#9149;
   // UNI[4052] := 16#6709;
   // UNI[4053] := 16#53CB;
   // UNI[4054] := 16#53F3;
   // UNI[4055] := 16#4F51;
   // UNI[4056] := 16#91C9;
   // UNI[4057] := 16#8BF1;
   // UNI[4058] := 16#53C8;
   // UNI[4059] := 16#5E7C;
   // UNI[4060] := 16#8FC2;
   // UNI[4061] := 16#6DE4;
   // UNI[4062] := 16#4E8E;
   // UNI[4063] := 16#76C2;
   // UNI[4064] := 16#6986;
   // UNI[4065] := 16#865E;
   // UNI[4066] := 16#611A;
   // UNI[4067] := 16#8206;
   // UNI[4068] := 16#4F59;
   // UNI[4069] := 16#4FDE;
   // UNI[4070] := 16#903E;
   // UNI[4071] := 16#9C7C;
   // UNI[4072] := 16#6109;
   // UNI[4073] := 16#6E1D;
   // UNI[4074] := 16#6E14;
   // UNI[4075] := 16#9685;
   // UNI[4076] := 16#4E88;
   // UNI[4077] := 16#5A31;
   // UNI[4078] := 16#96E8;
   // UNI[4079] := 16#4E0E;
   // UNI[4080] := 16#5C7F;
   // UNI[4081] := 16#79B9;
   // UNI[4082] := 16#5B87;
   // UNI[4083] := 16#8BED;
   // UNI[4084] := 16#7FBD;
   // UNI[4085] := 16#7389;
   // UNI[4086] := 16#57DF;
   // UNI[4087] := 16#828B;
   // UNI[4088] := 16#90C1;
   // UNI[4089] := 16#5401;
   // UNI[4090] := 16#9047;
   // UNI[4091] := 16#55BB;
   // UNI[4092] := 16#5CEA;
   // UNI[4093] := 16#5FA1;
   // UNI[4094] := 16#6108;
   // UNI[4095] := 16#6B32;
   // UNI[4096] := 16#72F1;
   // UNI[4097] := 16#80B2;
   // UNI[4098] := 16#8A89;
   // UNI[4099] := 16#6D74;
   // UNI[4100] := 16#5BD3;
   // UNI[4101] := 16#88D5;
   // UNI[4102] := 16#9884;
   // UNI[4103] := 16#8C6B;
   // UNI[4104] := 16#9A6D;
   // UNI[4105] := 16#9E33;
   // UNI[4106] := 16#6E0A;
   // UNI[4107] := 16#51A4;
   // UNI[4108] := 16#5143;
   // UNI[4109] := 16#57A3;
   // UNI[4110] := 16#8881;
   // UNI[4111] := 16#539F;
   // UNI[4112] := 16#63F4;
   // UNI[4113] := 16#8F95;
   // UNI[4114] := 16#56ED;
   // UNI[4115] := 16#5458;
   // UNI[4116] := 16#5706;
   // UNI[4117] := 16#733F;
   // UNI[4118] := 16#6E90;
   // UNI[4119] := 16#7F18;
   // UNI[4120] := 16#8FDC;
   // UNI[4121] := 16#82D1;
   // UNI[4122] := 16#613F;
   // UNI[4123] := 16#6028;
   // UNI[4124] := 16#9662;
   // UNI[4125] := 16#66F0;
   // UNI[4126] := 16#7EA6;
   // UNI[4127] := 16#8D8A;
   // UNI[4128] := 16#8DC3;
   // UNI[4129] := 16#94A5;
   // UNI[4130] := 16#5CB3;
   // UNI[4131] := 16#7CA4;
   // UNI[4132] := 16#6708;
   // UNI[4133] := 16#60A6;
   // UNI[4134] := 16#9605;
   // UNI[4135] := 16#8018;
   // UNI[4136] := 16#4E91;
   // UNI[4137] := 16#90E7;
   // UNI[4138] := 16#5300;
   // UNI[4139] := 16#9668;
   // UNI[4140] := 16#5141;
   // UNI[4141] := 16#8FD0;
   // UNI[4142] := 16#8574;
   // UNI[4143] := 16#915D;
   // UNI[4144] := 16#6655;
   // UNI[4145] := 16#97F5;
   // UNI[4146] := 16#5B55;
   // UNI[4147] := 16#531D;
   // UNI[4148] := 16#7838;
   // UNI[4149] := 16#6742;
   // UNI[4150] := 16#683D;
   // UNI[4151] := 16#54C9;
   // UNI[4152] := 16#707E;
   // UNI[4153] := 16#5BB0;
   // UNI[4154] := 16#8F7D;
   // UNI[4155] := 16#518D;
   // UNI[4156] := 16#5728;
   // UNI[4157] := 16#54B1;
   // UNI[4158] := 16#6512;
   // UNI[4159] := 16#6682;
   // UNI[4160] := 16#8D5E;
   // UNI[4161] := 16#8D43;
   // UNI[4162] := 16#810F;
   // UNI[4163] := 16#846C;
   // UNI[4164] := 16#906D;
   // UNI[4165] := 16#7CDF;
   // UNI[4166] := 16#51FF;
   // UNI[4167] := 16#85FB;
   // UNI[4168] := 16#67A3;
   // UNI[4169] := 16#65E9;
   // UNI[4170] := 16#6FA1;
   // UNI[4171] := 16#86A4;
   // UNI[4172] := 16#8E81;
   // UNI[4173] := 16#566A;
   // UNI[4174] := 16#9020;
   // UNI[4175] := 16#7682;
   // UNI[4176] := 16#7076;
   // UNI[4177] := 16#71E5;
   // UNI[4178] := 16#8D23;
   // UNI[4179] := 16#62E9;
   // UNI[4180] := 16#5219;
   // UNI[4181] := 16#6CFD;
   // UNI[4182] := 16#8D3C;
   // UNI[4183] := 16#600E;
   // UNI[4184] := 16#589E;
   // UNI[4185] := 16#618E;
   // UNI[4186] := 16#66FE;
   // UNI[4187] := 16#8D60;
   // UNI[4188] := 16#624E;
   // UNI[4189] := 16#55B3;
   // UNI[4190] := 16#6E23;
   // UNI[4191] := 16#672D;
   // UNI[4192] := 16#8F67;
   // UNI[4193] := 16#94E1;
   // UNI[4194] := 16#95F8;
   // UNI[4195] := 16#7728;
   // UNI[4196] := 16#6805;
   // UNI[4197] := 16#69A8;
   // UNI[4198] := 16#548B;
   // UNI[4199] := 16#4E4D;
   // UNI[4200] := 16#70B8;
   // UNI[4201] := 16#8BC8;
   // UNI[4202] := 16#6458;
   // UNI[4203] := 16#658B;
   // UNI[4204] := 16#5B85;
   // UNI[4205] := 16#7A84;
   // UNI[4206] := 16#503A;
   // UNI[4207] := 16#5BE8;
   // UNI[4208] := 16#77BB;
   // UNI[4209] := 16#6BE1;
   // UNI[4210] := 16#8A79;
   // UNI[4211] := 16#7C98;
   // UNI[4212] := 16#6CBE;
   // UNI[4213] := 16#76CF;
   // UNI[4214] := 16#65A9;
   // UNI[4215] := 16#8F97;
   // UNI[4216] := 16#5D2D;
   // UNI[4217] := 16#5C55;
   // UNI[4218] := 16#8638;
   // UNI[4219] := 16#6808;
   // UNI[4220] := 16#5360;
   // UNI[4221] := 16#6218;
   // UNI[4222] := 16#7AD9;
   // UNI[4223] := 16#6E5B;
   // UNI[4224] := 16#7EFD;
   // UNI[4225] := 16#6A1F;
   // UNI[4226] := 16#7AE0;
   // UNI[4227] := 16#5F70;
   // UNI[4228] := 16#6F33;
   // UNI[4229] := 16#5F20;
   // UNI[4230] := 16#638C;
   // UNI[4231] := 16#6DA8;
   // UNI[4232] := 16#6756;
   // UNI[4233] := 16#4E08;
   // UNI[4234] := 16#5E10;
   // UNI[4235] := 16#8D26;
   // UNI[4236] := 16#4ED7;
   // UNI[4237] := 16#80C0;
   // UNI[4238] := 16#7634;
   // UNI[4239] := 16#969C;
   // UNI[4240] := 16#62DB;
   // UNI[4241] := 16#662D;
   // UNI[4242] := 16#627E;
   // UNI[4243] := 16#6CBC;
   // UNI[4244] := 16#8D75;
   // UNI[4245] := 16#7167;
   // UNI[4246] := 16#7F69;
   // UNI[4247] := 16#5146;
   // UNI[4248] := 16#8087;
   // UNI[4249] := 16#53EC;
   // UNI[4250] := 16#906E;
   // UNI[4251] := 16#6298;
   // UNI[4252] := 16#54F2;
   // UNI[4253] := 16#86F0;
   // UNI[4254] := 16#8F99;
   // UNI[4255] := 16#8005;
   // UNI[4256] := 16#9517;
   // UNI[4257] := 16#8517;
   // UNI[4258] := 16#8FD9;
   // UNI[4259] := 16#6D59;
   // UNI[4260] := 16#73CD;
   // UNI[4261] := 16#659F;
   // UNI[4262] := 16#771F;
   // UNI[4263] := 16#7504;
   // UNI[4264] := 16#7827;
   // UNI[4265] := 16#81FB;
   // UNI[4266] := 16#8D1E;
   // UNI[4267] := 16#9488;
   // UNI[4268] := 16#4FA6;
   // UNI[4269] := 16#6795;
   // UNI[4270] := 16#75B9;
   // UNI[4271] := 16#8BCA;
   // UNI[4272] := 16#9707;
   // UNI[4273] := 16#632F;
   // UNI[4274] := 16#9547;
   // UNI[4275] := 16#9635;
   // UNI[4276] := 16#84B8;
   // UNI[4277] := 16#6323;
   // UNI[4278] := 16#7741;
   // UNI[4279] := 16#5F81;
   // UNI[4280] := 16#72F0;
   // UNI[4281] := 16#4E89;
   // UNI[4282] := 16#6014;
   // UNI[4283] := 16#6574;
   // UNI[4284] := 16#62EF;
   // UNI[4285] := 16#6B63;
   // UNI[4286] := 16#653F;
   // UNI[4287] := 16#5E27;
   // UNI[4288] := 16#75C7;
   // UNI[4289] := 16#90D1;
   // UNI[4290] := 16#8BC1;
   // UNI[4291] := 16#829D;
   // UNI[4292] := 16#679D;
   // UNI[4293] := 16#652F;
   // UNI[4294] := 16#5431;
   // UNI[4295] := 16#8718;
   // UNI[4296] := 16#77E5;
   // UNI[4297] := 16#80A2;
   // UNI[4298] := 16#8102;
   // UNI[4299] := 16#6C41;
   // UNI[4300] := 16#4E4B;
   // UNI[4301] := 16#7EC7;
   // UNI[4302] := 16#804C;
   // UNI[4303] := 16#76F4;
   // UNI[4304] := 16#690D;
   // UNI[4305] := 16#6B96;
   // UNI[4306] := 16#6267;
   // UNI[4307] := 16#503C;
   // UNI[4308] := 16#4F84;
   // UNI[4309] := 16#5740;
   // UNI[4310] := 16#6307;
   // UNI[4311] := 16#6B62;
   // UNI[4312] := 16#8DBE;
   // UNI[4313] := 16#53EA;
   // UNI[4314] := 16#65E8;
   // UNI[4315] := 16#7EB8;
   // UNI[4316] := 16#5FD7;
   // UNI[4317] := 16#631A;
   // UNI[4318] := 16#63B7;
   // UNI[4319] := 16#81F3;
   // UNI[4320] := 16#81F4;
   // UNI[4321] := 16#7F6E;
   // UNI[4322] := 16#5E1C;
   // UNI[4323] := 16#5CD9;
   // UNI[4324] := 16#5236;
   // UNI[4325] := 16#667A;
   // UNI[4326] := 16#79E9;
   // UNI[4327] := 16#7A1A;
   // UNI[4328] := 16#8D28;
   // UNI[4329] := 16#7099;
   // UNI[4330] := 16#75D4;
   // UNI[4331] := 16#6EDE;
   // UNI[4332] := 16#6CBB;
   // UNI[4333] := 16#7A92;
   // UNI[4334] := 16#4E2D;
   // UNI[4335] := 16#76C5;
   // UNI[4336] := 16#5FE0;
   // UNI[4337] := 16#949F;
   // UNI[4338] := 16#8877;
   // UNI[4339] := 16#7EC8;
   // UNI[4340] := 16#79CD;
   // UNI[4341] := 16#80BF;
   // UNI[4342] := 16#91CD;
   // UNI[4343] := 16#4EF2;
   // UNI[4344] := 16#4F17;
   // UNI[4345] := 16#821F;
   // UNI[4346] := 16#5468;
   // UNI[4347] := 16#5DDE;
   // UNI[4348] := 16#6D32;
   // UNI[4349] := 16#8BCC;
   // UNI[4350] := 16#7CA5;
   // UNI[4351] := 16#8F74;
   // UNI[4352] := 16#8098;
   // UNI[4353] := 16#5E1A;
   // UNI[4354] := 16#5492;
   // UNI[4355] := 16#76B1;
   // UNI[4356] := 16#5B99;
   // UNI[4357] := 16#663C;
   // UNI[4358] := 16#9AA4;
   // UNI[4359] := 16#73E0;
   // UNI[4360] := 16#682A;
   // UNI[4361] := 16#86DB;
   // UNI[4362] := 16#6731;
   // UNI[4363] := 16#732A;
   // UNI[4364] := 16#8BF8;
   // UNI[4365] := 16#8BDB;
   // UNI[4366] := 16#9010;
   // UNI[4367] := 16#7AF9;
   // UNI[4368] := 16#70DB;
   // UNI[4369] := 16#716E;
   // UNI[4370] := 16#62C4;
   // UNI[4371] := 16#77A9;
   // UNI[4372] := 16#5631;
   // UNI[4373] := 16#4E3B;
   // UNI[4374] := 16#8457;
   // UNI[4375] := 16#67F1;
   // UNI[4376] := 16#52A9;
   // UNI[4377] := 16#86C0;
   // UNI[4378] := 16#8D2E;
   // UNI[4379] := 16#94F8;
   // UNI[4380] := 16#7B51;
   // UNI[4381] := 16#4F4F;
   // UNI[4382] := 16#6CE8;
   // UNI[4383] := 16#795D;
   // UNI[4384] := 16#9A7B;
   // UNI[4385] := 16#6293;
   // UNI[4386] := 16#722A;
   // UNI[4387] := 16#62FD;
   // UNI[4388] := 16#4E13;
   // UNI[4389] := 16#7816;
   // UNI[4390] := 16#8F6C;
   // UNI[4391] := 16#64B0;
   // UNI[4392] := 16#8D5A;
   // UNI[4393] := 16#7BC6;
   // UNI[4394] := 16#6869;
   // UNI[4395] := 16#5E84;
   // UNI[4396] := 16#88C5;
   // UNI[4397] := 16#5986;
   // UNI[4398] := 16#649E;
   // UNI[4399] := 16#58EE;
   // UNI[4400] := 16#72B6;
   // UNI[4401] := 16#690E;
   // UNI[4402] := 16#9525;
   // UNI[4403] := 16#8FFD;
   // UNI[4404] := 16#8D58;
   // UNI[4405] := 16#5760;
   // UNI[4406] := 16#7F00;
   // UNI[4407] := 16#8C06;
   // UNI[4408] := 16#51C6;
   // UNI[4409] := 16#6349;
   // UNI[4410] := 16#62D9;
   // UNI[4411] := 16#5353;
   // UNI[4412] := 16#684C;
   // UNI[4413] := 16#7422;
   // UNI[4414] := 16#8301;
   // UNI[4415] := 16#914C;
   // UNI[4416] := 16#5544;
   // UNI[4417] := 16#7740;
   // UNI[4418] := 16#707C;
   // UNI[4419] := 16#6D4A;
   // UNI[4420] := 16#5179;
   // UNI[4421] := 16#54A8;
   // UNI[4422] := 16#8D44;
   // UNI[4423] := 16#59FF;
   // UNI[4424] := 16#6ECB;
   // UNI[4425] := 16#6DC4;
   // UNI[4426] := 16#5B5C;
   // UNI[4427] := 16#7D2B;
   // UNI[4428] := 16#4ED4;
   // UNI[4429] := 16#7C7D;
   // UNI[4430] := 16#6ED3;
   // UNI[4431] := 16#5B50;
   // UNI[4432] := 16#81EA;
   // UNI[4433] := 16#6E0D;
   // UNI[4434] := 16#5B57;
   // UNI[4435] := 16#9B03;
   // UNI[4436] := 16#68D5;
   // UNI[4437] := 16#8E2A;
   // UNI[4438] := 16#5B97;
   // UNI[4439] := 16#7EFC;
   // UNI[4440] := 16#603B;
   // UNI[4441] := 16#7EB5;
   // UNI[4442] := 16#90B9;
   // UNI[4443] := 16#8D70;
   // UNI[4444] := 16#594F;
   // UNI[4445] := 16#63CD;
   // UNI[4446] := 16#79DF;
   // UNI[4447] := 16#8DB3;
   // UNI[4448] := 16#5352;
   // UNI[4449] := 16#65CF;
   // UNI[4450] := 16#7956;
   // UNI[4451] := 16#8BC5;
   // UNI[4452] := 16#963B;
   // UNI[4453] := 16#7EC4;
   // UNI[4454] := 16#94BB;
   // UNI[4455] := 16#7E82;
   // UNI[4456] := 16#5634;
   // UNI[4457] := 16#9189;
   // UNI[4458] := 16#6700;
   // UNI[4459] := 16#7F6A;
   // UNI[4460] := 16#5C0A;
   // UNI[4461] := 16#9075;
   // UNI[4462] := 16#6628;
   // UNI[4463] := 16#5DE6;
   // UNI[4464] := 16#4F50;
   // UNI[4465] := 16#67DE;
   // UNI[4466] := 16#505A;
   // UNI[4467] := 16#4F5C;
   // UNI[4468] := 16#5750;
   // UNI[4469] := 16#5EA7;
   // UNI[4470] := 16#4E8D;
   // UNI[4471] := 16#4E0C;
   // UNI[4472] := 16#5140;
   // UNI[4473] := 16#4E10;
   // UNI[4474] := 16#5EFF;
   // UNI[4475] := 16#5345;
   // UNI[4476] := 16#4E15;
   // UNI[4477] := 16#4E98;
   // UNI[4478] := 16#4E1E;
   // UNI[4479] := 16#9B32;
   // UNI[4480] := 16#5B6C;
   // UNI[4481] := 16#5669;
   // UNI[4482] := 16#4E28;
   // UNI[4483] := 16#79BA;
   // UNI[4484] := 16#4E3F;
   // UNI[4485] := 16#5315;
   // UNI[4486] := 16#4E47;
   // UNI[4487] := 16#592D;
   // UNI[4488] := 16#723B;
   // UNI[4489] := 16#536E;
   // UNI[4490] := 16#6C10;
   // UNI[4491] := 16#56DF;
   // UNI[4492] := 16#80E4;
   // UNI[4493] := 16#9997;
   // UNI[4494] := 16#6BD3;
   // UNI[4495] := 16#777E;
   // UNI[4496] := 16#9F17;
   // UNI[4497] := 16#4E36;
   // UNI[4498] := 16#4E9F;
   // UNI[4499] := 16#9F10;
   // UNI[4500] := 16#4E5C;
   // UNI[4501] := 16#4E69;
   // UNI[4502] := 16#4E93;
   // UNI[4503] := 16#8288;
   // UNI[4504] := 16#5B5B;
   // UNI[4505] := 16#556C;
   // UNI[4506] := 16#560F;
   // UNI[4507] := 16#4EC4;
   // UNI[4508] := 16#538D;
   // UNI[4509] := 16#539D;
   // UNI[4510] := 16#53A3;
   // UNI[4511] := 16#53A5;
   // UNI[4512] := 16#53AE;
   // UNI[4513] := 16#9765;
   // UNI[4514] := 16#8D5D;
   // UNI[4515] := 16#531A;
   // UNI[4516] := 16#53F5;
   // UNI[4517] := 16#5326;
   // UNI[4518] := 16#532E;
   // UNI[4519] := 16#533E;
   // UNI[4520] := 16#8D5C;
   // UNI[4521] := 16#5366;
   // UNI[4522] := 16#5363;
   // UNI[4523] := 16#5202;
   // UNI[4524] := 16#5208;
   // UNI[4525] := 16#520E;
   // UNI[4526] := 16#522D;
   // UNI[4527] := 16#5233;
   // UNI[4528] := 16#523F;
   // UNI[4529] := 16#5240;
   // UNI[4530] := 16#524C;
   // UNI[4531] := 16#525E;
   // UNI[4532] := 16#5261;
   // UNI[4533] := 16#525C;
   // UNI[4534] := 16#84AF;
   // UNI[4535] := 16#527D;
   // UNI[4536] := 16#5282;
   // UNI[4537] := 16#5281;
   // UNI[4538] := 16#5290;
   // UNI[4539] := 16#5293;
   // UNI[4540] := 16#5182;
   // UNI[4541] := 16#7F54;
   // UNI[4542] := 16#4EBB;
   // UNI[4543] := 16#4EC3;
   // UNI[4544] := 16#4EC9;
   // UNI[4545] := 16#4EC2;
   // UNI[4546] := 16#4EE8;
   // UNI[4547] := 16#4EE1;
   // UNI[4548] := 16#4EEB;
   // UNI[4549] := 16#4EDE;
   // UNI[4550] := 16#4F1B;
   // UNI[4551] := 16#4EF3;
   // UNI[4552] := 16#4F22;
   // UNI[4553] := 16#4F64;
   // UNI[4554] := 16#4EF5;
   // UNI[4555] := 16#4F25;
   // UNI[4556] := 16#4F27;
   // UNI[4557] := 16#4F09;
   // UNI[4558] := 16#4F2B;
   // UNI[4559] := 16#4F5E;
   // UNI[4560] := 16#4F67;
   // UNI[4561] := 16#6538;
   // UNI[4562] := 16#4F5A;
   // UNI[4563] := 16#4F5D;
   // UNI[4564] := 16#4F5F;
   // UNI[4565] := 16#4F57;
   // UNI[4566] := 16#4F32;
   // UNI[4567] := 16#4F3D;
   // UNI[4568] := 16#4F76;
   // UNI[4569] := 16#4F74;
   // UNI[4570] := 16#4F91;
   // UNI[4571] := 16#4F89;
   // UNI[4572] := 16#4F83;
   // UNI[4573] := 16#4F8F;
   // UNI[4574] := 16#4F7E;
   // UNI[4575] := 16#4F7B;
   // UNI[4576] := 16#4FAA;
   // UNI[4577] := 16#4F7C;
   // UNI[4578] := 16#4FAC;
   // UNI[4579] := 16#4F94;
   // UNI[4580] := 16#4FE6;
   // UNI[4581] := 16#4FE8;
   // UNI[4582] := 16#4FEA;
   // UNI[4583] := 16#4FC5;
   // UNI[4584] := 16#4FDA;
   // UNI[4585] := 16#4FE3;
   // UNI[4586] := 16#4FDC;
   // UNI[4587] := 16#4FD1;
   // UNI[4588] := 16#4FDF;
   // UNI[4589] := 16#4FF8;
   // UNI[4590] := 16#5029;
   // UNI[4591] := 16#504C;
   // UNI[4592] := 16#4FF3;
   // UNI[4593] := 16#502C;
   // UNI[4594] := 16#500F;
   // UNI[4595] := 16#502E;
   // UNI[4596] := 16#502D;
   // UNI[4597] := 16#4FFE;
   // UNI[4598] := 16#501C;
   // UNI[4599] := 16#500C;
   // UNI[4600] := 16#5025;
   // UNI[4601] := 16#5028;
   // UNI[4602] := 16#507E;
   // UNI[4603] := 16#5043;
   // UNI[4604] := 16#5055;
   // UNI[4605] := 16#5048;
   // UNI[4606] := 16#504E;
   // UNI[4607] := 16#506C;
   // UNI[4608] := 16#507B;
   // UNI[4609] := 16#50A5;
   // UNI[4610] := 16#50A7;
   // UNI[4611] := 16#50A9;
   // UNI[4612] := 16#50BA;
   // UNI[4613] := 16#50D6;
   // UNI[4614] := 16#5106;
   // UNI[4615] := 16#50ED;
   // UNI[4616] := 16#50EC;
   // UNI[4617] := 16#50E6;
   // UNI[4618] := 16#50EE;
   // UNI[4619] := 16#5107;
   // UNI[4620] := 16#510B;
   // UNI[4621] := 16#4EDD;
   // UNI[4622] := 16#6C3D;
   // UNI[4623] := 16#4F58;
   // UNI[4624] := 16#4F65;
   // UNI[4625] := 16#4FCE;
   // UNI[4626] := 16#9FA0;
   // UNI[4627] := 16#6C46;
   // UNI[4628] := 16#7C74;
   // UNI[4629] := 16#516E;
   // UNI[4630] := 16#5DFD;
   // UNI[4631] := 16#9EC9;
   // UNI[4632] := 16#9998;
   // UNI[4633] := 16#5181;
   // UNI[4634] := 16#5914;
   // UNI[4635] := 16#52F9;
   // UNI[4636] := 16#530D;
   // UNI[4637] := 16#8A07;
   // UNI[4638] := 16#5310;
   // UNI[4639] := 16#51EB;
   // UNI[4640] := 16#5919;
   // UNI[4641] := 16#5155;
   // UNI[4642] := 16#4EA0;
   // UNI[4643] := 16#5156;
   // UNI[4644] := 16#4EB3;
   // UNI[4645] := 16#886E;
   // UNI[4646] := 16#88A4;
   // UNI[4647] := 16#4EB5;
   // UNI[4648] := 16#8114;
   // UNI[4649] := 16#88D2;
   // UNI[4650] := 16#7980;
   // UNI[4651] := 16#5B34;
   // UNI[4652] := 16#8803;
   // UNI[4653] := 16#7FB8;
   // UNI[4654] := 16#51AB;
   // UNI[4655] := 16#51B1;
   // UNI[4656] := 16#51BD;
   // UNI[4657] := 16#51BC;
   // UNI[4658] := 16#51C7;
   // UNI[4659] := 16#5196;
   // UNI[4660] := 16#51A2;
   // UNI[4661] := 16#51A5;
   // UNI[4662] := 16#8BA0;
   // UNI[4663] := 16#8BA6;
   // UNI[4664] := 16#8BA7;
   // UNI[4665] := 16#8BAA;
   // UNI[4666] := 16#8BB4;
   // UNI[4667] := 16#8BB5;
   // UNI[4668] := 16#8BB7;
   // UNI[4669] := 16#8BC2;
   // UNI[4670] := 16#8BC3;
   // UNI[4671] := 16#8BCB;
   // UNI[4672] := 16#8BCF;
   // UNI[4673] := 16#8BCE;
   // UNI[4674] := 16#8BD2;
   // UNI[4675] := 16#8BD3;
   // UNI[4676] := 16#8BD4;
   // UNI[4677] := 16#8BD6;
   // UNI[4678] := 16#8BD8;
   // UNI[4679] := 16#8BD9;
   // UNI[4680] := 16#8BDC;
   // UNI[4681] := 16#8BDF;
   // UNI[4682] := 16#8BE0;
   // UNI[4683] := 16#8BE4;
   // UNI[4684] := 16#8BE8;
   // UNI[4685] := 16#8BE9;
   // UNI[4686] := 16#8BEE;
   // UNI[4687] := 16#8BF0;
   // UNI[4688] := 16#8BF3;
   // UNI[4689] := 16#8BF6;
   // UNI[4690] := 16#8BF9;
   // UNI[4691] := 16#8BFC;
   // UNI[4692] := 16#8BFF;
   // UNI[4693] := 16#8C00;
   // UNI[4694] := 16#8C02;
   // UNI[4695] := 16#8C04;
   // UNI[4696] := 16#8C07;
   // UNI[4697] := 16#8C0C;
   // UNI[4698] := 16#8C0F;
   // UNI[4699] := 16#8C11;
   // UNI[4700] := 16#8C12;
   // UNI[4701] := 16#8C14;
   // UNI[4702] := 16#8C15;
   // UNI[4703] := 16#8C16;
   // UNI[4704] := 16#8C19;
   // UNI[4705] := 16#8C1B;
   // UNI[4706] := 16#8C18;
   // UNI[4707] := 16#8C1D;
   // UNI[4708] := 16#8C1F;
   // UNI[4709] := 16#8C20;
   // UNI[4710] := 16#8C21;
   // UNI[4711] := 16#8C25;
   // UNI[4712] := 16#8C27;
   // UNI[4713] := 16#8C2A;
   // UNI[4714] := 16#8C2B;
   // UNI[4715] := 16#8C2E;
   // UNI[4716] := 16#8C2F;
   // UNI[4717] := 16#8C32;
   // UNI[4718] := 16#8C33;
   // UNI[4719] := 16#8C35;
   // UNI[4720] := 16#8C36;
   // UNI[4721] := 16#5369;
   // UNI[4722] := 16#537A;
   // UNI[4723] := 16#961D;
   // UNI[4724] := 16#9622;
   // UNI[4725] := 16#9621;
   // UNI[4726] := 16#9631;
   // UNI[4727] := 16#962A;
   // UNI[4728] := 16#963D;
   // UNI[4729] := 16#963C;
   // UNI[4730] := 16#9642;
   // UNI[4731] := 16#9649;
   // UNI[4732] := 16#9654;
   // UNI[4733] := 16#965F;
   // UNI[4734] := 16#9667;
   // UNI[4735] := 16#966C;
   // UNI[4736] := 16#9672;
   // UNI[4737] := 16#9674;
   // UNI[4738] := 16#9688;
   // UNI[4739] := 16#968D;
   // UNI[4740] := 16#9697;
   // UNI[4741] := 16#96B0;
   // UNI[4742] := 16#9097;
   // UNI[4743] := 16#909B;
   // UNI[4744] := 16#909D;
   // UNI[4745] := 16#9099;
   // UNI[4746] := 16#90AC;
   // UNI[4747] := 16#90A1;
   // UNI[4748] := 16#90B4;
   // UNI[4749] := 16#90B3;
   // UNI[4750] := 16#90B6;
   // UNI[4751] := 16#90BA;
   // UNI[4752] := 16#90B8;
   // UNI[4753] := 16#90B0;
   // UNI[4754] := 16#90CF;
   // UNI[4755] := 16#90C5;
   // UNI[4756] := 16#90BE;
   // UNI[4757] := 16#90D0;
   // UNI[4758] := 16#90C4;
   // UNI[4759] := 16#90C7;
   // UNI[4760] := 16#90D3;
   // UNI[4761] := 16#90E6;
   // UNI[4762] := 16#90E2;
   // UNI[4763] := 16#90DC;
   // UNI[4764] := 16#90D7;
   // UNI[4765] := 16#90DB;
   // UNI[4766] := 16#90EB;
   // UNI[4767] := 16#90EF;
   // UNI[4768] := 16#90FE;
   // UNI[4769] := 16#9104;
   // UNI[4770] := 16#9122;
   // UNI[4771] := 16#911E;
   // UNI[4772] := 16#9123;
   // UNI[4773] := 16#9131;
   // UNI[4774] := 16#912F;
   // UNI[4775] := 16#9139;
   // UNI[4776] := 16#9143;
   // UNI[4777] := 16#9146;
   // UNI[4778] := 16#520D;
   // UNI[4779] := 16#5942;
   // UNI[4780] := 16#52A2;
   // UNI[4781] := 16#52AC;
   // UNI[4782] := 16#52AD;
   // UNI[4783] := 16#52BE;
   // UNI[4784] := 16#54FF;
   // UNI[4785] := 16#52D0;
   // UNI[4786] := 16#52D6;
   // UNI[4787] := 16#52F0;
   // UNI[4788] := 16#53DF;
   // UNI[4789] := 16#71EE;
   // UNI[4790] := 16#77CD;
   // UNI[4791] := 16#5EF4;
   // UNI[4792] := 16#51F5;
   // UNI[4793] := 16#51FC;
   // UNI[4794] := 16#9B2F;
   // UNI[4795] := 16#53B6;
   // UNI[4796] := 16#5F01;
   // UNI[4797] := 16#755A;
   // UNI[4798] := 16#5DEF;
   // UNI[4799] := 16#574C;
   // UNI[4800] := 16#57A9;
   // UNI[4801] := 16#57A1;
   // UNI[4802] := 16#587E;
   // UNI[4803] := 16#58BC;
   // UNI[4804] := 16#58C5;
   // UNI[4805] := 16#58D1;
   // UNI[4806] := 16#5729;
   // UNI[4807] := 16#572C;
   // UNI[4808] := 16#572A;
   // UNI[4809] := 16#5733;
   // UNI[4810] := 16#5739;
   // UNI[4811] := 16#572E;
   // UNI[4812] := 16#572F;
   // UNI[4813] := 16#575C;
   // UNI[4814] := 16#573B;
   // UNI[4815] := 16#5742;
   // UNI[4816] := 16#5769;
   // UNI[4817] := 16#5785;
   // UNI[4818] := 16#576B;
   // UNI[4819] := 16#5786;
   // UNI[4820] := 16#577C;
   // UNI[4821] := 16#577B;
   // UNI[4822] := 16#5768;
   // UNI[4823] := 16#576D;
   // UNI[4824] := 16#5776;
   // UNI[4825] := 16#5773;
   // UNI[4826] := 16#57AD;
   // UNI[4827] := 16#57A4;
   // UNI[4828] := 16#578C;
   // UNI[4829] := 16#57B2;
   // UNI[4830] := 16#57CF;
   // UNI[4831] := 16#57A7;
   // UNI[4832] := 16#57B4;
   // UNI[4833] := 16#5793;
   // UNI[4834] := 16#57A0;
   // UNI[4835] := 16#57D5;
   // UNI[4836] := 16#57D8;
   // UNI[4837] := 16#57DA;
   // UNI[4838] := 16#57D9;
   // UNI[4839] := 16#57D2;
   // UNI[4840] := 16#57B8;
   // UNI[4841] := 16#57F4;
   // UNI[4842] := 16#57EF;
   // UNI[4843] := 16#57F8;
   // UNI[4844] := 16#57E4;
   // UNI[4845] := 16#57DD;
   // UNI[4846] := 16#580B;
   // UNI[4847] := 16#580D;
   // UNI[4848] := 16#57FD;
   // UNI[4849] := 16#57ED;
   // UNI[4850] := 16#5800;
   // UNI[4851] := 16#581E;
   // UNI[4852] := 16#5819;
   // UNI[4853] := 16#5844;
   // UNI[4854] := 16#5820;
   // UNI[4855] := 16#5865;
   // UNI[4856] := 16#586C;
   // UNI[4857] := 16#5881;
   // UNI[4858] := 16#5889;
   // UNI[4859] := 16#589A;
   // UNI[4860] := 16#5880;
   // UNI[4861] := 16#99A8;
   // UNI[4862] := 16#9F19;
   // UNI[4863] := 16#61FF;
   // UNI[4864] := 16#8279;
   // UNI[4865] := 16#827D;
   // UNI[4866] := 16#827F;
   // UNI[4867] := 16#828F;
   // UNI[4868] := 16#828A;
   // UNI[4869] := 16#82A8;
   // UNI[4870] := 16#8284;
   // UNI[4871] := 16#828E;
   // UNI[4872] := 16#8291;
   // UNI[4873] := 16#8297;
   // UNI[4874] := 16#8299;
   // UNI[4875] := 16#82AB;
   // UNI[4876] := 16#82B8;
   // UNI[4877] := 16#82BE;
   // UNI[4878] := 16#82B0;
   // UNI[4879] := 16#82C8;
   // UNI[4880] := 16#82CA;
   // UNI[4881] := 16#82E3;
   // UNI[4882] := 16#8298;
   // UNI[4883] := 16#82B7;
   // UNI[4884] := 16#82AE;
   // UNI[4885] := 16#82CB;
   // UNI[4886] := 16#82CC;
   // UNI[4887] := 16#82C1;
   // UNI[4888] := 16#82A9;
   // UNI[4889] := 16#82B4;
   // UNI[4890] := 16#82A1;
   // UNI[4891] := 16#82AA;
   // UNI[4892] := 16#829F;
   // UNI[4893] := 16#82C4;
   // UNI[4894] := 16#82CE;
   // UNI[4895] := 16#82A4;
   // UNI[4896] := 16#82E1;
   // UNI[4897] := 16#8309;
   // UNI[4898] := 16#82F7;
   // UNI[4899] := 16#82E4;
   // UNI[4900] := 16#830F;
   // UNI[4901] := 16#8307;
   // UNI[4902] := 16#82DC;
   // UNI[4903] := 16#82F4;
   // UNI[4904] := 16#82D2;
   // UNI[4905] := 16#82D8;
   // UNI[4906] := 16#830C;
   // UNI[4907] := 16#82FB;
   // UNI[4908] := 16#82D3;
   // UNI[4909] := 16#8311;
   // UNI[4910] := 16#831A;
   // UNI[4911] := 16#8306;
   // UNI[4912] := 16#8314;
   // UNI[4913] := 16#8315;
   // UNI[4914] := 16#82E0;
   // UNI[4915] := 16#82D5;
   // UNI[4916] := 16#831C;
   // UNI[4917] := 16#8351;
   // UNI[4918] := 16#835B;
   // UNI[4919] := 16#835C;
   // UNI[4920] := 16#8308;
   // UNI[4921] := 16#8392;
   // UNI[4922] := 16#833C;
   // UNI[4923] := 16#8334;
   // UNI[4924] := 16#8331;
   // UNI[4925] := 16#839B;
   // UNI[4926] := 16#835E;
   // UNI[4927] := 16#832F;
   // UNI[4928] := 16#834F;
   // UNI[4929] := 16#8347;
   // UNI[4930] := 16#8343;
   // UNI[4931] := 16#835F;
   // UNI[4932] := 16#8340;
   // UNI[4933] := 16#8317;
   // UNI[4934] := 16#8360;
   // UNI[4935] := 16#832D;
   // UNI[4936] := 16#833A;
   // UNI[4937] := 16#8333;
   // UNI[4938] := 16#8366;
   // UNI[4939] := 16#8365;
   // UNI[4940] := 16#8368;
   // UNI[4941] := 16#831B;
   // UNI[4942] := 16#8369;
   // UNI[4943] := 16#836C;
   // UNI[4944] := 16#836A;
   // UNI[4945] := 16#836D;
   // UNI[4946] := 16#836E;
   // UNI[4947] := 16#83B0;
   // UNI[4948] := 16#8378;
   // UNI[4949] := 16#83B3;
   // UNI[4950] := 16#83B4;
   // UNI[4951] := 16#83A0;
   // UNI[4952] := 16#83AA;
   // UNI[4953] := 16#8393;
   // UNI[4954] := 16#839C;
   // UNI[4955] := 16#8385;
   // UNI[4956] := 16#837C;
   // UNI[4957] := 16#83B6;
   // UNI[4958] := 16#83A9;
   // UNI[4959] := 16#837D;
   // UNI[4960] := 16#83B8;
   // UNI[4961] := 16#837B;
   // UNI[4962] := 16#8398;
   // UNI[4963] := 16#839E;
   // UNI[4964] := 16#83A8;
   // UNI[4965] := 16#83BA;
   // UNI[4966] := 16#83BC;
   // UNI[4967] := 16#83C1;
   // UNI[4968] := 16#8401;
   // UNI[4969] := 16#83E5;
   // UNI[4970] := 16#83D8;
   // UNI[4971] := 16#5807;
   // UNI[4972] := 16#8418;
   // UNI[4973] := 16#840B;
   // UNI[4974] := 16#83DD;
   // UNI[4975] := 16#83FD;
   // UNI[4976] := 16#83D6;
   // UNI[4977] := 16#841C;
   // UNI[4978] := 16#8438;
   // UNI[4979] := 16#8411;
   // UNI[4980] := 16#8406;
   // UNI[4981] := 16#83D4;
   // UNI[4982] := 16#83DF;
   // UNI[4983] := 16#840F;
   // UNI[4984] := 16#8403;
   // UNI[4985] := 16#83F8;
   // UNI[4986] := 16#83F9;
   // UNI[4987] := 16#83EA;
   // UNI[4988] := 16#83C5;
   // UNI[4989] := 16#83C0;
   // UNI[4990] := 16#8426;
   // UNI[4991] := 16#83F0;
   // UNI[4992] := 16#83E1;
   // UNI[4993] := 16#845C;
   // UNI[4994] := 16#8451;
   // UNI[4995] := 16#845A;
   // UNI[4996] := 16#8459;
   // UNI[4997] := 16#8473;
   // UNI[4998] := 16#8487;
   // UNI[4999] := 16#8488;
   // UNI[5000] := 16#847A;
   // UNI[5001] := 16#8489;
   // UNI[5002] := 16#8478;
   // UNI[5003] := 16#843C;
   // UNI[5004] := 16#8446;
   // UNI[5005] := 16#8469;
   // UNI[5006] := 16#8476;
   // UNI[5007] := 16#848C;
   // UNI[5008] := 16#848E;
   // UNI[5009] := 16#8431;
   // UNI[5010] := 16#846D;
   // UNI[5011] := 16#84C1;
   // UNI[5012] := 16#84CD;
   // UNI[5013] := 16#84D0;
   // UNI[5014] := 16#84E6;
   // UNI[5015] := 16#84BD;
   // UNI[5016] := 16#84D3;
   // UNI[5017] := 16#84CA;
   // UNI[5018] := 16#84BF;
   // UNI[5019] := 16#84BA;
   // UNI[5020] := 16#84E0;
   // UNI[5021] := 16#84A1;
   // UNI[5022] := 16#84B9;
   // UNI[5023] := 16#84B4;
   // UNI[5024] := 16#8497;
   // UNI[5025] := 16#84E5;
   // UNI[5026] := 16#84E3;
   // UNI[5027] := 16#850C;
   // UNI[5028] := 16#750D;
   // UNI[5029] := 16#8538;
   // UNI[5030] := 16#84F0;
   // UNI[5031] := 16#8539;
   // UNI[5032] := 16#851F;
   // UNI[5033] := 16#853A;
   // UNI[5034] := 16#8556;
   // UNI[5035] := 16#853B;
   // UNI[5036] := 16#84FF;
   // UNI[5037] := 16#84FC;
   // UNI[5038] := 16#8559;
   // UNI[5039] := 16#8548;
   // UNI[5040] := 16#8568;
   // UNI[5041] := 16#8564;
   // UNI[5042] := 16#855E;
   // UNI[5043] := 16#857A;
   // UNI[5044] := 16#77A2;
   // UNI[5045] := 16#8543;
   // UNI[5046] := 16#8572;
   // UNI[5047] := 16#857B;
   // UNI[5048] := 16#85A4;
   // UNI[5049] := 16#85A8;
   // UNI[5050] := 16#8587;
   // UNI[5051] := 16#858F;
   // UNI[5052] := 16#8579;
   // UNI[5053] := 16#85AE;
   // UNI[5054] := 16#859C;
   // UNI[5055] := 16#8585;
   // UNI[5056] := 16#85B9;
   // UNI[5057] := 16#85B7;
   // UNI[5058] := 16#85B0;
   // UNI[5059] := 16#85D3;
   // UNI[5060] := 16#85C1;
   // UNI[5061] := 16#85DC;
   // UNI[5062] := 16#85FF;
   // UNI[5063] := 16#8627;
   // UNI[5064] := 16#8605;
   // UNI[5065] := 16#8629;
   // UNI[5066] := 16#8616;
   // UNI[5067] := 16#863C;
   // UNI[5068] := 16#5EFE;
   // UNI[5069] := 16#5F08;
   // UNI[5070] := 16#593C;
   // UNI[5071] := 16#5941;
   // UNI[5072] := 16#8037;
   // UNI[5073] := 16#5955;
   // UNI[5074] := 16#595A;
   // UNI[5075] := 16#5958;
   // UNI[5076] := 16#530F;
   // UNI[5077] := 16#5C22;
   // UNI[5078] := 16#5C25;
   // UNI[5079] := 16#5C2C;
   // UNI[5080] := 16#5C34;
   // UNI[5081] := 16#624C;
   // UNI[5082] := 16#626A;
   // UNI[5083] := 16#629F;
   // UNI[5084] := 16#62BB;
   // UNI[5085] := 16#62CA;
   // UNI[5086] := 16#62DA;
   // UNI[5087] := 16#62D7;
   // UNI[5088] := 16#62EE;
   // UNI[5089] := 16#6322;
   // UNI[5090] := 16#62F6;
   // UNI[5091] := 16#6339;
   // UNI[5092] := 16#634B;
   // UNI[5093] := 16#6343;
   // UNI[5094] := 16#63AD;
   // UNI[5095] := 16#63F6;
   // UNI[5096] := 16#6371;
   // UNI[5097] := 16#637A;
   // UNI[5098] := 16#638E;
   // UNI[5099] := 16#63B4;
   // UNI[5100] := 16#636D;
   // UNI[5101] := 16#63AC;
   // UNI[5102] := 16#638A;
   // UNI[5103] := 16#6369;
   // UNI[5104] := 16#63AE;
   // UNI[5105] := 16#63BC;
   // UNI[5106] := 16#63F2;
   // UNI[5107] := 16#63F8;
   // UNI[5108] := 16#63E0;
   // UNI[5109] := 16#63FF;
   // UNI[5110] := 16#63C4;
   // UNI[5111] := 16#63DE;
   // UNI[5112] := 16#63CE;
   // UNI[5113] := 16#6452;
   // UNI[5114] := 16#63C6;
   // UNI[5115] := 16#63BE;
   // UNI[5116] := 16#6445;
   // UNI[5117] := 16#6441;
   // UNI[5118] := 16#640B;
   // UNI[5119] := 16#641B;
   // UNI[5120] := 16#6420;
   // UNI[5121] := 16#640C;
   // UNI[5122] := 16#6426;
   // UNI[5123] := 16#6421;
   // UNI[5124] := 16#645E;
   // UNI[5125] := 16#6484;
   // UNI[5126] := 16#646D;
   // UNI[5127] := 16#6496;
   // UNI[5128] := 16#647A;
   // UNI[5129] := 16#64B7;
   // UNI[5130] := 16#64B8;
   // UNI[5131] := 16#6499;
   // UNI[5132] := 16#64BA;
   // UNI[5133] := 16#64C0;
   // UNI[5134] := 16#64D0;
   // UNI[5135] := 16#64D7;
   // UNI[5136] := 16#64E4;
   // UNI[5137] := 16#64E2;
   // UNI[5138] := 16#6509;
   // UNI[5139] := 16#6525;
   // UNI[5140] := 16#652E;
   // UNI[5141] := 16#5F0B;
   // UNI[5142] := 16#5FD2;
   // UNI[5143] := 16#7519;
   // UNI[5144] := 16#5F11;
   // UNI[5145] := 16#535F;
   // UNI[5146] := 16#53F1;
   // UNI[5147] := 16#53FD;
   // UNI[5148] := 16#53E9;
   // UNI[5149] := 16#53E8;
   // UNI[5150] := 16#53FB;
   // UNI[5151] := 16#5412;
   // UNI[5152] := 16#5416;
   // UNI[5153] := 16#5406;
   // UNI[5154] := 16#544B;
   // UNI[5155] := 16#5452;
   // UNI[5156] := 16#5453;
   // UNI[5157] := 16#5454;
   // UNI[5158] := 16#5456;
   // UNI[5159] := 16#5443;
   // UNI[5160] := 16#5421;
   // UNI[5161] := 16#5457;
   // UNI[5162] := 16#5459;
   // UNI[5163] := 16#5423;
   // UNI[5164] := 16#5432;
   // UNI[5165] := 16#5482;
   // UNI[5166] := 16#5494;
   // UNI[5167] := 16#5477;
   // UNI[5168] := 16#5471;
   // UNI[5169] := 16#5464;
   // UNI[5170] := 16#549A;
   // UNI[5171] := 16#549B;
   // UNI[5172] := 16#5484;
   // UNI[5173] := 16#5476;
   // UNI[5174] := 16#5466;
   // UNI[5175] := 16#549D;
   // UNI[5176] := 16#54D0;
   // UNI[5177] := 16#54AD;
   // UNI[5178] := 16#54C2;
   // UNI[5179] := 16#54B4;
   // UNI[5180] := 16#54D2;
   // UNI[5181] := 16#54A7;
   // UNI[5182] := 16#54A6;
   // UNI[5183] := 16#54D3;
   // UNI[5184] := 16#54D4;
   // UNI[5185] := 16#5472;
   // UNI[5186] := 16#54A3;
   // UNI[5187] := 16#54D5;
   // UNI[5188] := 16#54BB;
   // UNI[5189] := 16#54BF;
   // UNI[5190] := 16#54CC;
   // UNI[5191] := 16#54D9;
   // UNI[5192] := 16#54DA;
   // UNI[5193] := 16#54DC;
   // UNI[5194] := 16#54A9;
   // UNI[5195] := 16#54AA;
   // UNI[5196] := 16#54A4;
   // UNI[5197] := 16#54DD;
   // UNI[5198] := 16#54CF;
   // UNI[5199] := 16#54DE;
   // UNI[5200] := 16#551B;
   // UNI[5201] := 16#54E7;
   // UNI[5202] := 16#5520;
   // UNI[5203] := 16#54FD;
   // UNI[5204] := 16#5514;
   // UNI[5205] := 16#54F3;
   // UNI[5206] := 16#5522;
   // UNI[5207] := 16#5523;
   // UNI[5208] := 16#550F;
   // UNI[5209] := 16#5511;
   // UNI[5210] := 16#5527;
   // UNI[5211] := 16#552A;
   // UNI[5212] := 16#5567;
   // UNI[5213] := 16#558F;
   // UNI[5214] := 16#55B5;
   // UNI[5215] := 16#5549;
   // UNI[5216] := 16#556D;
   // UNI[5217] := 16#5541;
   // UNI[5218] := 16#5555;
   // UNI[5219] := 16#553F;
   // UNI[5220] := 16#5550;
   // UNI[5221] := 16#553C;
   // UNI[5222] := 16#5537;
   // UNI[5223] := 16#5556;
   // UNI[5224] := 16#5575;
   // UNI[5225] := 16#5576;
   // UNI[5226] := 16#5577;
   // UNI[5227] := 16#5533;
   // UNI[5228] := 16#5530;
   // UNI[5229] := 16#555C;
   // UNI[5230] := 16#558B;
   // UNI[5231] := 16#55D2;
   // UNI[5232] := 16#5583;
   // UNI[5233] := 16#55B1;
   // UNI[5234] := 16#55B9;
   // UNI[5235] := 16#5588;
   // UNI[5236] := 16#5581;
   // UNI[5237] := 16#559F;
   // UNI[5238] := 16#557E;
   // UNI[5239] := 16#55D6;
   // UNI[5240] := 16#5591;
   // UNI[5241] := 16#557B;
   // UNI[5242] := 16#55DF;
   // UNI[5243] := 16#55BD;
   // UNI[5244] := 16#55BE;
   // UNI[5245] := 16#5594;
   // UNI[5246] := 16#5599;
   // UNI[5247] := 16#55EA;
   // UNI[5248] := 16#55F7;
   // UNI[5249] := 16#55C9;
   // UNI[5250] := 16#561F;
   // UNI[5251] := 16#55D1;
   // UNI[5252] := 16#55EB;
   // UNI[5253] := 16#55EC;
   // UNI[5254] := 16#55D4;
   // UNI[5255] := 16#55E6;
   // UNI[5256] := 16#55DD;
   // UNI[5257] := 16#55C4;
   // UNI[5258] := 16#55EF;
   // UNI[5259] := 16#55E5;
   // UNI[5260] := 16#55F2;
   // UNI[5261] := 16#55F3;
   // UNI[5262] := 16#55CC;
   // UNI[5263] := 16#55CD;
   // UNI[5264] := 16#55E8;
   // UNI[5265] := 16#55F5;
   // UNI[5266] := 16#55E4;
   // UNI[5267] := 16#8F94;
   // UNI[5268] := 16#561E;
   // UNI[5269] := 16#5608;
   // UNI[5270] := 16#560C;
   // UNI[5271] := 16#5601;
   // UNI[5272] := 16#5624;
   // UNI[5273] := 16#5623;
   // UNI[5274] := 16#55FE;
   // UNI[5275] := 16#5600;
   // UNI[5276] := 16#5627;
   // UNI[5277] := 16#562D;
   // UNI[5278] := 16#5658;
   // UNI[5279] := 16#5639;
   // UNI[5280] := 16#5657;
   // UNI[5281] := 16#562C;
   // UNI[5282] := 16#564D;
   // UNI[5283] := 16#5662;
   // UNI[5284] := 16#5659;
   // UNI[5285] := 16#565C;
   // UNI[5286] := 16#564C;
   // UNI[5287] := 16#5654;
   // UNI[5288] := 16#5686;
   // UNI[5289] := 16#5664;
   // UNI[5290] := 16#5671;
   // UNI[5291] := 16#566B;
   // UNI[5292] := 16#567B;
   // UNI[5293] := 16#567C;
   // UNI[5294] := 16#5685;
   // UNI[5295] := 16#5693;
   // UNI[5296] := 16#56AF;
   // UNI[5297] := 16#56D4;
   // UNI[5298] := 16#56D7;
   // UNI[5299] := 16#56DD;
   // UNI[5300] := 16#56E1;
   // UNI[5301] := 16#56F5;
   // UNI[5302] := 16#56EB;
   // UNI[5303] := 16#56F9;
   // UNI[5304] := 16#56FF;
   // UNI[5305] := 16#5704;
   // UNI[5306] := 16#570A;
   // UNI[5307] := 16#5709;
   // UNI[5308] := 16#571C;
   // UNI[5309] := 16#5E0F;
   // UNI[5310] := 16#5E19;
   // UNI[5311] := 16#5E14;
   // UNI[5312] := 16#5E11;
   // UNI[5313] := 16#5E31;
   // UNI[5314] := 16#5E3B;
   // UNI[5315] := 16#5E3C;
   // UNI[5316] := 16#5E37;
   // UNI[5317] := 16#5E44;
   // UNI[5318] := 16#5E54;
   // UNI[5319] := 16#5E5B;
   // UNI[5320] := 16#5E5E;
   // UNI[5321] := 16#5E61;
   // UNI[5322] := 16#5C8C;
   // UNI[5323] := 16#5C7A;
   // UNI[5324] := 16#5C8D;
   // UNI[5325] := 16#5C90;
   // UNI[5326] := 16#5C96;
   // UNI[5327] := 16#5C88;
   // UNI[5328] := 16#5C98;
   // UNI[5329] := 16#5C99;
   // UNI[5330] := 16#5C91;
   // UNI[5331] := 16#5C9A;
   // UNI[5332] := 16#5C9C;
   // UNI[5333] := 16#5CB5;
   // UNI[5334] := 16#5CA2;
   // UNI[5335] := 16#5CBD;
   // UNI[5336] := 16#5CAC;
   // UNI[5337] := 16#5CAB;
   // UNI[5338] := 16#5CB1;
   // UNI[5339] := 16#5CA3;
   // UNI[5340] := 16#5CC1;
   // UNI[5341] := 16#5CB7;
   // UNI[5342] := 16#5CC4;
   // UNI[5343] := 16#5CD2;
   // UNI[5344] := 16#5CE4;
   // UNI[5345] := 16#5CCB;
   // UNI[5346] := 16#5CE5;
   // UNI[5347] := 16#5D02;
   // UNI[5348] := 16#5D03;
   // UNI[5349] := 16#5D27;
   // UNI[5350] := 16#5D26;
   // UNI[5351] := 16#5D2E;
   // UNI[5352] := 16#5D24;
   // UNI[5353] := 16#5D1E;
   // UNI[5354] := 16#5D06;
   // UNI[5355] := 16#5D1B;
   // UNI[5356] := 16#5D58;
   // UNI[5357] := 16#5D3E;
   // UNI[5358] := 16#5D34;
   // UNI[5359] := 16#5D3D;
   // UNI[5360] := 16#5D6C;
   // UNI[5361] := 16#5D5B;
   // UNI[5362] := 16#5D6F;
   // UNI[5363] := 16#5D5D;
   // UNI[5364] := 16#5D6B;
   // UNI[5365] := 16#5D4B;
   // UNI[5366] := 16#5D4A;
   // UNI[5367] := 16#5D69;
   // UNI[5368] := 16#5D74;
   // UNI[5369] := 16#5D82;
   // UNI[5370] := 16#5D99;
   // UNI[5371] := 16#5D9D;
   // UNI[5372] := 16#8C73;
   // UNI[5373] := 16#5DB7;
   // UNI[5374] := 16#5DC5;
   // UNI[5375] := 16#5F73;
   // UNI[5376] := 16#5F77;
   // UNI[5377] := 16#5F82;
   // UNI[5378] := 16#5F87;
   // UNI[5379] := 16#5F89;
   // UNI[5380] := 16#5F8C;
   // UNI[5381] := 16#5F95;
   // UNI[5382] := 16#5F99;
   // UNI[5383] := 16#5F9C;
   // UNI[5384] := 16#5FA8;
   // UNI[5385] := 16#5FAD;
   // UNI[5386] := 16#5FB5;
   // UNI[5387] := 16#5FBC;
   // UNI[5388] := 16#8862;
   // UNI[5389] := 16#5F61;
   // UNI[5390] := 16#72AD;
   // UNI[5391] := 16#72B0;
   // UNI[5392] := 16#72B4;
   // UNI[5393] := 16#72B7;
   // UNI[5394] := 16#72B8;
   // UNI[5395] := 16#72C3;
   // UNI[5396] := 16#72C1;
   // UNI[5397] := 16#72CE;
   // UNI[5398] := 16#72CD;
   // UNI[5399] := 16#72D2;
   // UNI[5400] := 16#72E8;
   // UNI[5401] := 16#72EF;
   // UNI[5402] := 16#72E9;
   // UNI[5403] := 16#72F2;
   // UNI[5404] := 16#72F4;
   // UNI[5405] := 16#72F7;
   // UNI[5406] := 16#7301;
   // UNI[5407] := 16#72F3;
   // UNI[5408] := 16#7303;
   // UNI[5409] := 16#72FA;
   // UNI[5410] := 16#72FB;
   // UNI[5411] := 16#7317;
   // UNI[5412] := 16#7313;
   // UNI[5413] := 16#7321;
   // UNI[5414] := 16#730A;
   // UNI[5415] := 16#731E;
   // UNI[5416] := 16#731D;
   // UNI[5417] := 16#7315;
   // UNI[5418] := 16#7322;
   // UNI[5419] := 16#7339;
   // UNI[5420] := 16#7325;
   // UNI[5421] := 16#732C;
   // UNI[5422] := 16#7338;
   // UNI[5423] := 16#7331;
   // UNI[5424] := 16#7350;
   // UNI[5425] := 16#734D;
   // UNI[5426] := 16#7357;
   // UNI[5427] := 16#7360;
   // UNI[5428] := 16#736C;
   // UNI[5429] := 16#736F;
   // UNI[5430] := 16#737E;
   // UNI[5431] := 16#821B;
   // UNI[5432] := 16#5925;
   // UNI[5433] := 16#98E7;
   // UNI[5434] := 16#5924;
   // UNI[5435] := 16#5902;
   // UNI[5436] := 16#9963;
   // UNI[5437] := 16#9967;
   // UNI[5438] := 16#9968;
   // UNI[5439] := 16#9969;
   // UNI[5440] := 16#996A;
   // UNI[5441] := 16#996B;
   // UNI[5442] := 16#996C;
   // UNI[5443] := 16#9974;
   // UNI[5444] := 16#9977;
   // UNI[5445] := 16#997D;
   // UNI[5446] := 16#9980;
   // UNI[5447] := 16#9984;
   // UNI[5448] := 16#9987;
   // UNI[5449] := 16#998A;
   // UNI[5450] := 16#998D;
   // UNI[5451] := 16#9990;
   // UNI[5452] := 16#9991;
   // UNI[5453] := 16#9993;
   // UNI[5454] := 16#9994;
   // UNI[5455] := 16#9995;
   // UNI[5456] := 16#5E80;
   // UNI[5457] := 16#5E91;
   // UNI[5458] := 16#5E8B;
   // UNI[5459] := 16#5E96;
   // UNI[5460] := 16#5EA5;
   // UNI[5461] := 16#5EA0;
   // UNI[5462] := 16#5EB9;
   // UNI[5463] := 16#5EB5;
   // UNI[5464] := 16#5EBE;
   // UNI[5465] := 16#5EB3;
   // UNI[5466] := 16#8D53;
   // UNI[5467] := 16#5ED2;
   // UNI[5468] := 16#5ED1;
   // UNI[5469] := 16#5EDB;
   // UNI[5470] := 16#5EE8;
   // UNI[5471] := 16#5EEA;
   // UNI[5472] := 16#81BA;
   // UNI[5473] := 16#5FC4;
   // UNI[5474] := 16#5FC9;
   // UNI[5475] := 16#5FD6;
   // UNI[5476] := 16#5FCF;
   // UNI[5477] := 16#6003;
   // UNI[5478] := 16#5FEE;
   // UNI[5479] := 16#6004;
   // UNI[5480] := 16#5FE1;
   // UNI[5481] := 16#5FE4;
   // UNI[5482] := 16#5FFE;
   // UNI[5483] := 16#6005;
   // UNI[5484] := 16#6006;
   // UNI[5485] := 16#5FEA;
   // UNI[5486] := 16#5FED;
   // UNI[5487] := 16#5FF8;
   // UNI[5488] := 16#6019;
   // UNI[5489] := 16#6035;
   // UNI[5490] := 16#6026;
   // UNI[5491] := 16#601B;
   // UNI[5492] := 16#600F;
   // UNI[5493] := 16#600D;
   // UNI[5494] := 16#6029;
   // UNI[5495] := 16#602B;
   // UNI[5496] := 16#600A;
   // UNI[5497] := 16#603F;
   // UNI[5498] := 16#6021;
   // UNI[5499] := 16#6078;
   // UNI[5500] := 16#6079;
   // UNI[5501] := 16#607B;
   // UNI[5502] := 16#607A;
   // UNI[5503] := 16#6042;
   // UNI[5504] := 16#606A;
   // UNI[5505] := 16#607D;
   // UNI[5506] := 16#6096;
   // UNI[5507] := 16#609A;
   // UNI[5508] := 16#60AD;
   // UNI[5509] := 16#609D;
   // UNI[5510] := 16#6083;
   // UNI[5511] := 16#6092;
   // UNI[5512] := 16#608C;
   // UNI[5513] := 16#609B;
   // UNI[5514] := 16#60EC;
   // UNI[5515] := 16#60BB;
   // UNI[5516] := 16#60B1;
   // UNI[5517] := 16#60DD;
   // UNI[5518] := 16#60D8;
   // UNI[5519] := 16#60C6;
   // UNI[5520] := 16#60DA;
   // UNI[5521] := 16#60B4;
   // UNI[5522] := 16#6120;
   // UNI[5523] := 16#6126;
   // UNI[5524] := 16#6115;
   // UNI[5525] := 16#6123;
   // UNI[5526] := 16#60F4;
   // UNI[5527] := 16#6100;
   // UNI[5528] := 16#610E;
   // UNI[5529] := 16#612B;
   // UNI[5530] := 16#614A;
   // UNI[5531] := 16#6175;
   // UNI[5532] := 16#61AC;
   // UNI[5533] := 16#6194;
   // UNI[5534] := 16#61A7;
   // UNI[5535] := 16#61B7;
   // UNI[5536] := 16#61D4;
   // UNI[5537] := 16#61F5;
   // UNI[5538] := 16#5FDD;
   // UNI[5539] := 16#96B3;
   // UNI[5540] := 16#95E9;
   // UNI[5541] := 16#95EB;
   // UNI[5542] := 16#95F1;
   // UNI[5543] := 16#95F3;
   // UNI[5544] := 16#95F5;
   // UNI[5545] := 16#95F6;
   // UNI[5546] := 16#95FC;
   // UNI[5547] := 16#95FE;
   // UNI[5548] := 16#9603;
   // UNI[5549] := 16#9604;
   // UNI[5550] := 16#9606;
   // UNI[5551] := 16#9608;
   // UNI[5552] := 16#960A;
   // UNI[5553] := 16#960B;
   // UNI[5554] := 16#960C;
   // UNI[5555] := 16#960D;
   // UNI[5556] := 16#960F;
   // UNI[5557] := 16#9612;
   // UNI[5558] := 16#9615;
   // UNI[5559] := 16#9616;
   // UNI[5560] := 16#9617;
   // UNI[5561] := 16#9619;
   // UNI[5562] := 16#961A;
   // UNI[5563] := 16#4E2C;
   // UNI[5564] := 16#723F;
   // UNI[5565] := 16#6215;
   // UNI[5566] := 16#6C35;
   // UNI[5567] := 16#6C54;
   // UNI[5568] := 16#6C5C;
   // UNI[5569] := 16#6C4A;
   // UNI[5570] := 16#6CA3;
   // UNI[5571] := 16#6C85;
   // UNI[5572] := 16#6C90;
   // UNI[5573] := 16#6C94;
   // UNI[5574] := 16#6C8C;
   // UNI[5575] := 16#6C68;
   // UNI[5576] := 16#6C69;
   // UNI[5577] := 16#6C74;
   // UNI[5578] := 16#6C76;
   // UNI[5579] := 16#6C86;
   // UNI[5580] := 16#6CA9;
   // UNI[5581] := 16#6CD0;
   // UNI[5582] := 16#6CD4;
   // UNI[5583] := 16#6CAD;
   // UNI[5584] := 16#6CF7;
   // UNI[5585] := 16#6CF8;
   // UNI[5586] := 16#6CF1;
   // UNI[5587] := 16#6CD7;
   // UNI[5588] := 16#6CB2;
   // UNI[5589] := 16#6CE0;
   // UNI[5590] := 16#6CD6;
   // UNI[5591] := 16#6CFA;
   // UNI[5592] := 16#6CEB;
   // UNI[5593] := 16#6CEE;
   // UNI[5594] := 16#6CB1;
   // UNI[5595] := 16#6CD3;
   // UNI[5596] := 16#6CEF;
   // UNI[5597] := 16#6CFE;
   // UNI[5598] := 16#6D39;
   // UNI[5599] := 16#6D27;
   // UNI[5600] := 16#6D0C;
   // UNI[5601] := 16#6D43;
   // UNI[5602] := 16#6D48;
   // UNI[5603] := 16#6D07;
   // UNI[5604] := 16#6D04;
   // UNI[5605] := 16#6D19;
   // UNI[5606] := 16#6D0E;
   // UNI[5607] := 16#6D2B;
   // UNI[5608] := 16#6D4D;
   // UNI[5609] := 16#6D2E;
   // UNI[5610] := 16#6D35;
   // UNI[5611] := 16#6D1A;
   // UNI[5612] := 16#6D4F;
   // UNI[5613] := 16#6D52;
   // UNI[5614] := 16#6D54;
   // UNI[5615] := 16#6D33;
   // UNI[5616] := 16#6D91;
   // UNI[5617] := 16#6D6F;
   // UNI[5618] := 16#6D9E;
   // UNI[5619] := 16#6DA0;
   // UNI[5620] := 16#6D5E;
   // UNI[5621] := 16#6D93;
   // UNI[5622] := 16#6D94;
   // UNI[5623] := 16#6D5C;
   // UNI[5624] := 16#6D60;
   // UNI[5625] := 16#6D7C;
   // UNI[5626] := 16#6D63;
   // UNI[5627] := 16#6E1A;
   // UNI[5628] := 16#6DC7;
   // UNI[5629] := 16#6DC5;
   // UNI[5630] := 16#6DDE;
   // UNI[5631] := 16#6E0E;
   // UNI[5632] := 16#6DBF;
   // UNI[5633] := 16#6DE0;
   // UNI[5634] := 16#6E11;
   // UNI[5635] := 16#6DE6;
   // UNI[5636] := 16#6DDD;
   // UNI[5637] := 16#6DD9;
   // UNI[5638] := 16#6E16;
   // UNI[5639] := 16#6DAB;
   // UNI[5640] := 16#6E0C;
   // UNI[5641] := 16#6DAE;
   // UNI[5642] := 16#6E2B;
   // UNI[5643] := 16#6E6E;
   // UNI[5644] := 16#6E4E;
   // UNI[5645] := 16#6E6B;
   // UNI[5646] := 16#6EB2;
   // UNI[5647] := 16#6E5F;
   // UNI[5648] := 16#6E86;
   // UNI[5649] := 16#6E53;
   // UNI[5650] := 16#6E54;
   // UNI[5651] := 16#6E32;
   // UNI[5652] := 16#6E25;
   // UNI[5653] := 16#6E44;
   // UNI[5654] := 16#6EDF;
   // UNI[5655] := 16#6EB1;
   // UNI[5656] := 16#6E98;
   // UNI[5657] := 16#6EE0;
   // UNI[5658] := 16#6F2D;
   // UNI[5659] := 16#6EE2;
   // UNI[5660] := 16#6EA5;
   // UNI[5661] := 16#6EA7;
   // UNI[5662] := 16#6EBD;
   // UNI[5663] := 16#6EBB;
   // UNI[5664] := 16#6EB7;
   // UNI[5665] := 16#6ED7;
   // UNI[5666] := 16#6EB4;
   // UNI[5667] := 16#6ECF;
   // UNI[5668] := 16#6E8F;
   // UNI[5669] := 16#6EC2;
   // UNI[5670] := 16#6E9F;
   // UNI[5671] := 16#6F62;
   // UNI[5672] := 16#6F46;
   // UNI[5673] := 16#6F47;
   // UNI[5674] := 16#6F24;
   // UNI[5675] := 16#6F15;
   // UNI[5676] := 16#6EF9;
   // UNI[5677] := 16#6F2F;
   // UNI[5678] := 16#6F36;
   // UNI[5679] := 16#6F4B;
   // UNI[5680] := 16#6F74;
   // UNI[5681] := 16#6F2A;
   // UNI[5682] := 16#6F09;
   // UNI[5683] := 16#6F29;
   // UNI[5684] := 16#6F89;
   // UNI[5685] := 16#6F8D;
   // UNI[5686] := 16#6F8C;
   // UNI[5687] := 16#6F78;
   // UNI[5688] := 16#6F72;
   // UNI[5689] := 16#6F7C;
   // UNI[5690] := 16#6F7A;
   // UNI[5691] := 16#6FD1;
   // UNI[5692] := 16#6FC9;
   // UNI[5693] := 16#6FA7;
   // UNI[5694] := 16#6FB9;
   // UNI[5695] := 16#6FB6;
   // UNI[5696] := 16#6FC2;
   // UNI[5697] := 16#6FE1;
   // UNI[5698] := 16#6FEE;
   // UNI[5699] := 16#6FDE;
   // UNI[5700] := 16#6FE0;
   // UNI[5701] := 16#6FEF;
   // UNI[5702] := 16#701A;
   // UNI[5703] := 16#7023;
   // UNI[5704] := 16#701B;
   // UNI[5705] := 16#7039;
   // UNI[5706] := 16#7035;
   // UNI[5707] := 16#704F;
   // UNI[5708] := 16#705E;
   // UNI[5709] := 16#5B80;
   // UNI[5710] := 16#5B84;
   // UNI[5711] := 16#5B95;
   // UNI[5712] := 16#5B93;
   // UNI[5713] := 16#5BA5;
   // UNI[5714] := 16#5BB8;
   // UNI[5715] := 16#752F;
   // UNI[5716] := 16#9A9E;
   // UNI[5717] := 16#6434;
   // UNI[5718] := 16#5BE4;
   // UNI[5719] := 16#5BEE;
   // UNI[5720] := 16#8930;
   // UNI[5721] := 16#5BF0;
   // UNI[5722] := 16#8E47;
   // UNI[5723] := 16#8B07;
   // UNI[5724] := 16#8FB6;
   // UNI[5725] := 16#8FD3;
   // UNI[5726] := 16#8FD5;
   // UNI[5727] := 16#8FE5;
   // UNI[5728] := 16#8FEE;
   // UNI[5729] := 16#8FE4;
   // UNI[5730] := 16#8FE9;
   // UNI[5731] := 16#8FE6;
   // UNI[5732] := 16#8FF3;
   // UNI[5733] := 16#8FE8;
   // UNI[5734] := 16#9005;
   // UNI[5735] := 16#9004;
   // UNI[5736] := 16#900B;
   // UNI[5737] := 16#9026;
   // UNI[5738] := 16#9011;
   // UNI[5739] := 16#900D;
   // UNI[5740] := 16#9016;
   // UNI[5741] := 16#9021;
   // UNI[5742] := 16#9035;
   // UNI[5743] := 16#9036;
   // UNI[5744] := 16#902D;
   // UNI[5745] := 16#902F;
   // UNI[5746] := 16#9044;
   // UNI[5747] := 16#9051;
   // UNI[5748] := 16#9052;
   // UNI[5749] := 16#9050;
   // UNI[5750] := 16#9068;
   // UNI[5751] := 16#9058;
   // UNI[5752] := 16#9062;
   // UNI[5753] := 16#905B;
   // UNI[5754] := 16#66B9;
   // UNI[5755] := 16#9074;
   // UNI[5756] := 16#907D;
   // UNI[5757] := 16#9082;
   // UNI[5758] := 16#9088;
   // UNI[5759] := 16#9083;
   // UNI[5760] := 16#908B;
   // UNI[5761] := 16#5F50;
   // UNI[5762] := 16#5F57;
   // UNI[5763] := 16#5F56;
   // UNI[5764] := 16#5F58;
   // UNI[5765] := 16#5C3B;
   // UNI[5766] := 16#54AB;
   // UNI[5767] := 16#5C50;
   // UNI[5768] := 16#5C59;
   // UNI[5769] := 16#5B71;
   // UNI[5770] := 16#5C63;
   // UNI[5771] := 16#5C66;
   // UNI[5772] := 16#7FBC;
   // UNI[5773] := 16#5F2A;
   // UNI[5774] := 16#5F29;
   // UNI[5775] := 16#5F2D;
   // UNI[5776] := 16#8274;
   // UNI[5777] := 16#5F3C;
   // UNI[5778] := 16#9B3B;
   // UNI[5779] := 16#5C6E;
   // UNI[5780] := 16#5981;
   // UNI[5781] := 16#5983;
   // UNI[5782] := 16#598D;
   // UNI[5783] := 16#59A9;
   // UNI[5784] := 16#59AA;
   // UNI[5785] := 16#59A3;
   // UNI[5786] := 16#5997;
   // UNI[5787] := 16#59CA;
   // UNI[5788] := 16#59AB;
   // UNI[5789] := 16#599E;
   // UNI[5790] := 16#59A4;
   // UNI[5791] := 16#59D2;
   // UNI[5792] := 16#59B2;
   // UNI[5793] := 16#59AF;
   // UNI[5794] := 16#59D7;
   // UNI[5795] := 16#59BE;
   // UNI[5796] := 16#5A05;
   // UNI[5797] := 16#5A06;
   // UNI[5798] := 16#59DD;
   // UNI[5799] := 16#5A08;
   // UNI[5800] := 16#59E3;
   // UNI[5801] := 16#59D8;
   // UNI[5802] := 16#59F9;
   // UNI[5803] := 16#5A0C;
   // UNI[5804] := 16#5A09;
   // UNI[5805] := 16#5A32;
   // UNI[5806] := 16#5A34;
   // UNI[5807] := 16#5A11;
   // UNI[5808] := 16#5A23;
   // UNI[5809] := 16#5A13;
   // UNI[5810] := 16#5A40;
   // UNI[5811] := 16#5A67;
   // UNI[5812] := 16#5A4A;
   // UNI[5813] := 16#5A55;
   // UNI[5814] := 16#5A3C;
   // UNI[5815] := 16#5A62;
   // UNI[5816] := 16#5A75;
   // UNI[5817] := 16#80EC;
   // UNI[5818] := 16#5AAA;
   // UNI[5819] := 16#5A9B;
   // UNI[5820] := 16#5A77;
   // UNI[5821] := 16#5A7A;
   // UNI[5822] := 16#5ABE;
   // UNI[5823] := 16#5AEB;
   // UNI[5824] := 16#5AB2;
   // UNI[5825] := 16#5AD2;
   // UNI[5826] := 16#5AD4;
   // UNI[5827] := 16#5AB8;
   // UNI[5828] := 16#5AE0;
   // UNI[5829] := 16#5AE3;
   // UNI[5830] := 16#5AF1;
   // UNI[5831] := 16#5AD6;
   // UNI[5832] := 16#5AE6;
   // UNI[5833] := 16#5AD8;
   // UNI[5834] := 16#5ADC;
   // UNI[5835] := 16#5B09;
   // UNI[5836] := 16#5B17;
   // UNI[5837] := 16#5B16;
   // UNI[5838] := 16#5B32;
   // UNI[5839] := 16#5B37;
   // UNI[5840] := 16#5B40;
   // UNI[5841] := 16#5C15;
   // UNI[5842] := 16#5C1C;
   // UNI[5843] := 16#5B5A;
   // UNI[5844] := 16#5B65;
   // UNI[5845] := 16#5B73;
   // UNI[5846] := 16#5B51;
   // UNI[5847] := 16#5B53;
   // UNI[5848] := 16#5B62;
   // UNI[5849] := 16#9A75;
   // UNI[5850] := 16#9A77;
   // UNI[5851] := 16#9A78;
   // UNI[5852] := 16#9A7A;
   // UNI[5853] := 16#9A7F;
   // UNI[5854] := 16#9A7D;
   // UNI[5855] := 16#9A80;
   // UNI[5856] := 16#9A81;
   // UNI[5857] := 16#9A85;
   // UNI[5858] := 16#9A88;
   // UNI[5859] := 16#9A8A;
   // UNI[5860] := 16#9A90;
   // UNI[5861] := 16#9A92;
   // UNI[5862] := 16#9A93;
   // UNI[5863] := 16#9A96;
   // UNI[5864] := 16#9A98;
   // UNI[5865] := 16#9A9B;
   // UNI[5866] := 16#9A9C;
   // UNI[5867] := 16#9A9D;
   // UNI[5868] := 16#9A9F;
   // UNI[5869] := 16#9AA0;
   // UNI[5870] := 16#9AA2;
   // UNI[5871] := 16#9AA3;
   // UNI[5872] := 16#9AA5;
   // UNI[5873] := 16#9AA7;
   // UNI[5874] := 16#7E9F;
   // UNI[5875] := 16#7EA1;
   // UNI[5876] := 16#7EA3;
   // UNI[5877] := 16#7EA5;
   // UNI[5878] := 16#7EA8;
   // UNI[5879] := 16#7EA9;
   // UNI[5880] := 16#7EAD;
   // UNI[5881] := 16#7EB0;
   // UNI[5882] := 16#7EBE;
   // UNI[5883] := 16#7EC0;
   // UNI[5884] := 16#7EC1;
   // UNI[5885] := 16#7EC2;
   // UNI[5886] := 16#7EC9;
   // UNI[5887] := 16#7ECB;
   // UNI[5888] := 16#7ECC;
   // UNI[5889] := 16#7ED0;
   // UNI[5890] := 16#7ED4;
   // UNI[5891] := 16#7ED7;
   // UNI[5892] := 16#7EDB;
   // UNI[5893] := 16#7EE0;
   // UNI[5894] := 16#7EE1;
   // UNI[5895] := 16#7EE8;
   // UNI[5896] := 16#7EEB;
   // UNI[5897] := 16#7EEE;
   // UNI[5898] := 16#7EEF;
   // UNI[5899] := 16#7EF1;
   // UNI[5900] := 16#7EF2;
   // UNI[5901] := 16#7F0D;
   // UNI[5902] := 16#7EF6;
   // UNI[5903] := 16#7EFA;
   // UNI[5904] := 16#7EFB;
   // UNI[5905] := 16#7EFE;
   // UNI[5906] := 16#7F01;
   // UNI[5907] := 16#7F02;
   // UNI[5908] := 16#7F03;
   // UNI[5909] := 16#7F07;
   // UNI[5910] := 16#7F08;
   // UNI[5911] := 16#7F0B;
   // UNI[5912] := 16#7F0C;
   // UNI[5913] := 16#7F0F;
   // UNI[5914] := 16#7F11;
   // UNI[5915] := 16#7F12;
   // UNI[5916] := 16#7F17;
   // UNI[5917] := 16#7F19;
   // UNI[5918] := 16#7F1C;
   // UNI[5919] := 16#7F1B;
   // UNI[5920] := 16#7F1F;
   // UNI[5921] := 16#7F21;
   // UNI[5922] := 16#7F22;
   // UNI[5923] := 16#7F23;
   // UNI[5924] := 16#7F24;
   // UNI[5925] := 16#7F25;
   // UNI[5926] := 16#7F26;
   // UNI[5927] := 16#7F27;
   // UNI[5928] := 16#7F2A;
   // UNI[5929] := 16#7F2B;
   // UNI[5930] := 16#7F2C;
   // UNI[5931] := 16#7F2D;
   // UNI[5932] := 16#7F2F;
   // UNI[5933] := 16#7F30;
   // UNI[5934] := 16#7F31;
   // UNI[5935] := 16#7F32;
   // UNI[5936] := 16#7F33;
   // UNI[5937] := 16#7F35;
   // UNI[5938] := 16#5E7A;
   // UNI[5939] := 16#757F;
   // UNI[5940] := 16#5DDB;
   // UNI[5941] := 16#753E;
   // UNI[5942] := 16#9095;
   // UNI[5943] := 16#738E;
   // UNI[5944] := 16#7391;
   // UNI[5945] := 16#73AE;
   // UNI[5946] := 16#73A2;
   // UNI[5947] := 16#739F;
   // UNI[5948] := 16#73CF;
   // UNI[5949] := 16#73C2;
   // UNI[5950] := 16#73D1;
   // UNI[5951] := 16#73B7;
   // UNI[5952] := 16#73B3;
   // UNI[5953] := 16#73C0;
   // UNI[5954] := 16#73C9;
   // UNI[5955] := 16#73C8;
   // UNI[5956] := 16#73E5;
   // UNI[5957] := 16#73D9;
   // UNI[5958] := 16#987C;
   // UNI[5959] := 16#740A;
   // UNI[5960] := 16#73E9;
   // UNI[5961] := 16#73E7;
   // UNI[5962] := 16#73DE;
   // UNI[5963] := 16#73BA;
   // UNI[5964] := 16#73F2;
   // UNI[5965] := 16#740F;
   // UNI[5966] := 16#742A;
   // UNI[5967] := 16#745B;
   // UNI[5968] := 16#7426;
   // UNI[5969] := 16#7425;
   // UNI[5970] := 16#7428;
   // UNI[5971] := 16#7430;
   // UNI[5972] := 16#742E;
   // UNI[5973] := 16#742C;
   // UNI[5974] := 16#741B;
   // UNI[5975] := 16#741A;
   // UNI[5976] := 16#7441;
   // UNI[5977] := 16#745C;
   // UNI[5978] := 16#7457;
   // UNI[5979] := 16#7455;
   // UNI[5980] := 16#7459;
   // UNI[5981] := 16#7477;
   // UNI[5982] := 16#746D;
   // UNI[5983] := 16#747E;
   // UNI[5984] := 16#749C;
   // UNI[5985] := 16#748E;
   // UNI[5986] := 16#7480;
   // UNI[5987] := 16#7481;
   // UNI[5988] := 16#7487;
   // UNI[5989] := 16#748B;
   // UNI[5990] := 16#749E;
   // UNI[5991] := 16#74A8;
   // UNI[5992] := 16#74A9;
   // UNI[5993] := 16#7490;
   // UNI[5994] := 16#74A7;
   // UNI[5995] := 16#74D2;
   // UNI[5996] := 16#74BA;
   // UNI[5997] := 16#97EA;
   // UNI[5998] := 16#97EB;
   // UNI[5999] := 16#97EC;
   // UNI[6000] := 16#674C;
   // UNI[6001] := 16#6753;
   // UNI[6002] := 16#675E;
   // UNI[6003] := 16#6748;
   // UNI[6004] := 16#6769;
   // UNI[6005] := 16#67A5;
   // UNI[6006] := 16#6787;
   // UNI[6007] := 16#676A;
   // UNI[6008] := 16#6773;
   // UNI[6009] := 16#6798;
   // UNI[6010] := 16#67A7;
   // UNI[6011] := 16#6775;
   // UNI[6012] := 16#67A8;
   // UNI[6013] := 16#679E;
   // UNI[6014] := 16#67AD;
   // UNI[6015] := 16#678B;
   // UNI[6016] := 16#6777;
   // UNI[6017] := 16#677C;
   // UNI[6018] := 16#67F0;
   // UNI[6019] := 16#6809;
   // UNI[6020] := 16#67D8;
   // UNI[6021] := 16#680A;
   // UNI[6022] := 16#67E9;
   // UNI[6023] := 16#67B0;
   // UNI[6024] := 16#680C;
   // UNI[6025] := 16#67D9;
   // UNI[6026] := 16#67B5;
   // UNI[6027] := 16#67DA;
   // UNI[6028] := 16#67B3;
   // UNI[6029] := 16#67DD;
   // UNI[6030] := 16#6800;
   // UNI[6031] := 16#67C3;
   // UNI[6032] := 16#67B8;
   // UNI[6033] := 16#67E2;
   // UNI[6034] := 16#680E;
   // UNI[6035] := 16#67C1;
   // UNI[6036] := 16#67FD;
   // UNI[6037] := 16#6832;
   // UNI[6038] := 16#6833;
   // UNI[6039] := 16#6860;
   // UNI[6040] := 16#6861;
   // UNI[6041] := 16#684E;
   // UNI[6042] := 16#6862;
   // UNI[6043] := 16#6844;
   // UNI[6044] := 16#6864;
   // UNI[6045] := 16#6883;
   // UNI[6046] := 16#681D;
   // UNI[6047] := 16#6855;
   // UNI[6048] := 16#6866;
   // UNI[6049] := 16#6841;
   // UNI[6050] := 16#6867;
   // UNI[6051] := 16#6840;
   // UNI[6052] := 16#683E;
   // UNI[6053] := 16#684A;
   // UNI[6054] := 16#6849;
   // UNI[6055] := 16#6829;
   // UNI[6056] := 16#68B5;
   // UNI[6057] := 16#688F;
   // UNI[6058] := 16#6874;
   // UNI[6059] := 16#6877;
   // UNI[6060] := 16#6893;
   // UNI[6061] := 16#686B;
   // UNI[6062] := 16#68C2;
   // UNI[6063] := 16#696E;
   // UNI[6064] := 16#68FC;
   // UNI[6065] := 16#691F;
   // UNI[6066] := 16#6920;
   // UNI[6067] := 16#68F9;
   // UNI[6068] := 16#6924;
   // UNI[6069] := 16#68F0;
   // UNI[6070] := 16#690B;
   // UNI[6071] := 16#6901;
   // UNI[6072] := 16#6957;
   // UNI[6073] := 16#68E3;
   // UNI[6074] := 16#6910;
   // UNI[6075] := 16#6971;
   // UNI[6076] := 16#6939;
   // UNI[6077] := 16#6960;
   // UNI[6078] := 16#6942;
   // UNI[6079] := 16#695D;
   // UNI[6080] := 16#6984;
   // UNI[6081] := 16#696B;
   // UNI[6082] := 16#6980;
   // UNI[6083] := 16#6998;
   // UNI[6084] := 16#6978;
   // UNI[6085] := 16#6934;
   // UNI[6086] := 16#69CC;
   // UNI[6087] := 16#6987;
   // UNI[6088] := 16#6988;
   // UNI[6089] := 16#69CE;
   // UNI[6090] := 16#6989;
   // UNI[6091] := 16#6966;
   // UNI[6092] := 16#6963;
   // UNI[6093] := 16#6979;
   // UNI[6094] := 16#699B;
   // UNI[6095] := 16#69A7;
   // UNI[6096] := 16#69BB;
   // UNI[6097] := 16#69AB;
   // UNI[6098] := 16#69AD;
   // UNI[6099] := 16#69D4;
   // UNI[6100] := 16#69B1;
   // UNI[6101] := 16#69C1;
   // UNI[6102] := 16#69CA;
   // UNI[6103] := 16#69DF;
   // UNI[6104] := 16#6995;
   // UNI[6105] := 16#69E0;
   // UNI[6106] := 16#698D;
   // UNI[6107] := 16#69FF;
   // UNI[6108] := 16#6A2F;
   // UNI[6109] := 16#69ED;
   // UNI[6110] := 16#6A17;
   // UNI[6111] := 16#6A18;
   // UNI[6112] := 16#6A65;
   // UNI[6113] := 16#69F2;
   // UNI[6114] := 16#6A44;
   // UNI[6115] := 16#6A3E;
   // UNI[6116] := 16#6AA0;
   // UNI[6117] := 16#6A50;
   // UNI[6118] := 16#6A5B;
   // UNI[6119] := 16#6A35;
   // UNI[6120] := 16#6A8E;
   // UNI[6121] := 16#6A79;
   // UNI[6122] := 16#6A3D;
   // UNI[6123] := 16#6A28;
   // UNI[6124] := 16#6A58;
   // UNI[6125] := 16#6A7C;
   // UNI[6126] := 16#6A91;
   // UNI[6127] := 16#6A90;
   // UNI[6128] := 16#6AA9;
   // UNI[6129] := 16#6A97;
   // UNI[6130] := 16#6AAB;
   // UNI[6131] := 16#7337;
   // UNI[6132] := 16#7352;
   // UNI[6133] := 16#6B81;
   // UNI[6134] := 16#6B82;
   // UNI[6135] := 16#6B87;
   // UNI[6136] := 16#6B84;
   // UNI[6137] := 16#6B92;
   // UNI[6138] := 16#6B93;
   // UNI[6139] := 16#6B8D;
   // UNI[6140] := 16#6B9A;
   // UNI[6141] := 16#6B9B;
   // UNI[6142] := 16#6BA1;
   // UNI[6143] := 16#6BAA;
   // UNI[6144] := 16#8F6B;
   // UNI[6145] := 16#8F6D;
   // UNI[6146] := 16#8F71;
   // UNI[6147] := 16#8F72;
   // UNI[6148] := 16#8F73;
   // UNI[6149] := 16#8F75;
   // UNI[6150] := 16#8F76;
   // UNI[6151] := 16#8F78;
   // UNI[6152] := 16#8F77;
   // UNI[6153] := 16#8F79;
   // UNI[6154] := 16#8F7A;
   // UNI[6155] := 16#8F7C;
   // UNI[6156] := 16#8F7E;
   // UNI[6157] := 16#8F81;
   // UNI[6158] := 16#8F82;
   // UNI[6159] := 16#8F84;
   // UNI[6160] := 16#8F87;
   // UNI[6161] := 16#8F8B;
   // UNI[6162] := 16#8F8D;
   // UNI[6163] := 16#8F8E;
   // UNI[6164] := 16#8F8F;
   // UNI[6165] := 16#8F98;
   // UNI[6166] := 16#8F9A;
   // UNI[6167] := 16#8ECE;
   // UNI[6168] := 16#620B;
   // UNI[6169] := 16#6217;
   // UNI[6170] := 16#621B;
   // UNI[6171] := 16#621F;
   // UNI[6172] := 16#6222;
   // UNI[6173] := 16#6221;
   // UNI[6174] := 16#6225;
   // UNI[6175] := 16#6224;
   // UNI[6176] := 16#622C;
   // UNI[6177] := 16#81E7;
   // UNI[6178] := 16#74EF;
   // UNI[6179] := 16#74F4;
   // UNI[6180] := 16#74FF;
   // UNI[6181] := 16#750F;
   // UNI[6182] := 16#7511;
   // UNI[6183] := 16#7513;
   // UNI[6184] := 16#6534;
   // UNI[6185] := 16#65EE;
   // UNI[6186] := 16#65EF;
   // UNI[6187] := 16#65F0;
   // UNI[6188] := 16#660A;
   // UNI[6189] := 16#6619;
   // UNI[6190] := 16#6772;
   // UNI[6191] := 16#6603;
   // UNI[6192] := 16#6615;
   // UNI[6193] := 16#6600;
   // UNI[6194] := 16#7085;
   // UNI[6195] := 16#66F7;
   // UNI[6196] := 16#661D;
   // UNI[6197] := 16#6634;
   // UNI[6198] := 16#6631;
   // UNI[6199] := 16#6636;
   // UNI[6200] := 16#6635;
   // UNI[6201] := 16#8006;
   // UNI[6202] := 16#665F;
   // UNI[6203] := 16#6654;
   // UNI[6204] := 16#6641;
   // UNI[6205] := 16#664F;
   // UNI[6206] := 16#6656;
   // UNI[6207] := 16#6661;
   // UNI[6208] := 16#6657;
   // UNI[6209] := 16#6677;
   // UNI[6210] := 16#6684;
   // UNI[6211] := 16#668C;
   // UNI[6212] := 16#66A7;
   // UNI[6213] := 16#669D;
   // UNI[6214] := 16#66BE;
   // UNI[6215] := 16#66DB;
   // UNI[6216] := 16#66DC;
   // UNI[6217] := 16#66E6;
   // UNI[6218] := 16#66E9;
   // UNI[6219] := 16#8D32;
   // UNI[6220] := 16#8D33;
   // UNI[6221] := 16#8D36;
   // UNI[6222] := 16#8D3B;
   // UNI[6223] := 16#8D3D;
   // UNI[6224] := 16#8D40;
   // UNI[6225] := 16#8D45;
   // UNI[6226] := 16#8D46;
   // UNI[6227] := 16#8D48;
   // UNI[6228] := 16#8D49;
   // UNI[6229] := 16#8D47;
   // UNI[6230] := 16#8D4D;
   // UNI[6231] := 16#8D55;
   // UNI[6232] := 16#8D59;
   // UNI[6233] := 16#89C7;
   // UNI[6234] := 16#89CA;
   // UNI[6235] := 16#89CB;
   // UNI[6236] := 16#89CC;
   // UNI[6237] := 16#89CE;
   // UNI[6238] := 16#89CF;
   // UNI[6239] := 16#89D0;
   // UNI[6240] := 16#89D1;
   // UNI[6241] := 16#726E;
   // UNI[6242] := 16#729F;
   // UNI[6243] := 16#725D;
   // UNI[6244] := 16#7266;
   // UNI[6245] := 16#726F;
   // UNI[6246] := 16#727E;
   // UNI[6247] := 16#727F;
   // UNI[6248] := 16#7284;
   // UNI[6249] := 16#728B;
   // UNI[6250] := 16#728D;
   // UNI[6251] := 16#728F;
   // UNI[6252] := 16#7292;
   // UNI[6253] := 16#6308;
   // UNI[6254] := 16#6332;
   // UNI[6255] := 16#63B0;
   // UNI[6256] := 16#643F;
   // UNI[6257] := 16#64D8;
   // UNI[6258] := 16#8004;
   // UNI[6259] := 16#6BEA;
   // UNI[6260] := 16#6BF3;
   // UNI[6261] := 16#6BFD;
   // UNI[6262] := 16#6BF5;
   // UNI[6263] := 16#6BF9;
   // UNI[6264] := 16#6C05;
   // UNI[6265] := 16#6C07;
   // UNI[6266] := 16#6C06;
   // UNI[6267] := 16#6C0D;
   // UNI[6268] := 16#6C15;
   // UNI[6269] := 16#6C18;
   // UNI[6270] := 16#6C19;
   // UNI[6271] := 16#6C1A;
   // UNI[6272] := 16#6C21;
   // UNI[6273] := 16#6C29;
   // UNI[6274] := 16#6C24;
   // UNI[6275] := 16#6C2A;
   // UNI[6276] := 16#6C32;
   // UNI[6277] := 16#6535;
   // UNI[6278] := 16#6555;
   // UNI[6279] := 16#656B;
   // UNI[6280] := 16#724D;
   // UNI[6281] := 16#7252;
   // UNI[6282] := 16#7256;
   // UNI[6283] := 16#7230;
   // UNI[6284] := 16#8662;
   // UNI[6285] := 16#5216;
   // UNI[6286] := 16#809F;
   // UNI[6287] := 16#809C;
   // UNI[6288] := 16#8093;
   // UNI[6289] := 16#80BC;
   // UNI[6290] := 16#670A;
   // UNI[6291] := 16#80BD;
   // UNI[6292] := 16#80B1;
   // UNI[6293] := 16#80AB;
   // UNI[6294] := 16#80AD;
   // UNI[6295] := 16#80B4;
   // UNI[6296] := 16#80B7;
   // UNI[6297] := 16#80E7;
   // UNI[6298] := 16#80E8;
   // UNI[6299] := 16#80E9;
   // UNI[6300] := 16#80EA;
   // UNI[6301] := 16#80DB;
   // UNI[6302] := 16#80C2;
   // UNI[6303] := 16#80C4;
   // UNI[6304] := 16#80D9;
   // UNI[6305] := 16#80CD;
   // UNI[6306] := 16#80D7;
   // UNI[6307] := 16#6710;
   // UNI[6308] := 16#80DD;
   // UNI[6309] := 16#80EB;
   // UNI[6310] := 16#80F1;
   // UNI[6311] := 16#80F4;
   // UNI[6312] := 16#80ED;
   // UNI[6313] := 16#810D;
   // UNI[6314] := 16#810E;
   // UNI[6315] := 16#80F2;
   // UNI[6316] := 16#80FC;
   // UNI[6317] := 16#6715;
   // UNI[6318] := 16#8112;
   // UNI[6319] := 16#8C5A;
   // UNI[6320] := 16#8136;
   // UNI[6321] := 16#811E;
   // UNI[6322] := 16#812C;
   // UNI[6323] := 16#8118;
   // UNI[6324] := 16#8132;
   // UNI[6325] := 16#8148;
   // UNI[6326] := 16#814C;
   // UNI[6327] := 16#8153;
   // UNI[6328] := 16#8174;
   // UNI[6329] := 16#8159;
   // UNI[6330] := 16#815A;
   // UNI[6331] := 16#8171;
   // UNI[6332] := 16#8160;
   // UNI[6333] := 16#8169;
   // UNI[6334] := 16#817C;
   // UNI[6335] := 16#817D;
   // UNI[6336] := 16#816D;
   // UNI[6337] := 16#8167;
   // UNI[6338] := 16#584D;
   // UNI[6339] := 16#5AB5;
   // UNI[6340] := 16#8188;
   // UNI[6341] := 16#8182;
   // UNI[6342] := 16#8191;
   // UNI[6343] := 16#6ED5;
   // UNI[6344] := 16#81A3;
   // UNI[6345] := 16#81AA;
   // UNI[6346] := 16#81CC;
   // UNI[6347] := 16#6726;
   // UNI[6348] := 16#81CA;
   // UNI[6349] := 16#81BB;
   // UNI[6350] := 16#81C1;
   // UNI[6351] := 16#81A6;
   // UNI[6352] := 16#6B24;
   // UNI[6353] := 16#6B37;
   // UNI[6354] := 16#6B39;
   // UNI[6355] := 16#6B43;
   // UNI[6356] := 16#6B46;
   // UNI[6357] := 16#6B59;
   // UNI[6358] := 16#98D1;
   // UNI[6359] := 16#98D2;
   // UNI[6360] := 16#98D3;
   // UNI[6361] := 16#98D5;
   // UNI[6362] := 16#98D9;
   // UNI[6363] := 16#98DA;
   // UNI[6364] := 16#6BB3;
   // UNI[6365] := 16#5F40;
   // UNI[6366] := 16#6BC2;
   // UNI[6367] := 16#89F3;
   // UNI[6368] := 16#6590;
   // UNI[6369] := 16#9F51;
   // UNI[6370] := 16#6593;
   // UNI[6371] := 16#65BC;
   // UNI[6372] := 16#65C6;
   // UNI[6373] := 16#65C4;
   // UNI[6374] := 16#65C3;
   // UNI[6375] := 16#65CC;
   // UNI[6376] := 16#65CE;
   // UNI[6377] := 16#65D2;
   // UNI[6378] := 16#65D6;
   // UNI[6379] := 16#7080;
   // UNI[6380] := 16#709C;
   // UNI[6381] := 16#7096;
   // UNI[6382] := 16#709D;
   // UNI[6383] := 16#70BB;
   // UNI[6384] := 16#70C0;
   // UNI[6385] := 16#70B7;
   // UNI[6386] := 16#70AB;
   // UNI[6387] := 16#70B1;
   // UNI[6388] := 16#70E8;
   // UNI[6389] := 16#70CA;
   // UNI[6390] := 16#7110;
   // UNI[6391] := 16#7113;
   // UNI[6392] := 16#7116;
   // UNI[6393] := 16#712F;
   // UNI[6394] := 16#7131;
   // UNI[6395] := 16#7173;
   // UNI[6396] := 16#715C;
   // UNI[6397] := 16#7168;
   // UNI[6398] := 16#7145;
   // UNI[6399] := 16#7172;
   // UNI[6400] := 16#714A;
   // UNI[6401] := 16#7178;
   // UNI[6402] := 16#717A;
   // UNI[6403] := 16#7198;
   // UNI[6404] := 16#71B3;
   // UNI[6405] := 16#71B5;
   // UNI[6406] := 16#71A8;
   // UNI[6407] := 16#71A0;
   // UNI[6408] := 16#71E0;
   // UNI[6409] := 16#71D4;
   // UNI[6410] := 16#71E7;
   // UNI[6411] := 16#71F9;
   // UNI[6412] := 16#721D;
   // UNI[6413] := 16#7228;
   // UNI[6414] := 16#706C;
   // UNI[6415] := 16#7118;
   // UNI[6416] := 16#7166;
   // UNI[6417] := 16#71B9;
   // UNI[6418] := 16#623E;
   // UNI[6419] := 16#623D;
   // UNI[6420] := 16#6243;
   // UNI[6421] := 16#6248;
   // UNI[6422] := 16#6249;
   // UNI[6423] := 16#793B;
   // UNI[6424] := 16#7940;
   // UNI[6425] := 16#7946;
   // UNI[6426] := 16#7949;
   // UNI[6427] := 16#795B;
   // UNI[6428] := 16#795C;
   // UNI[6429] := 16#7953;
   // UNI[6430] := 16#795A;
   // UNI[6431] := 16#7962;
   // UNI[6432] := 16#7957;
   // UNI[6433] := 16#7960;
   // UNI[6434] := 16#796F;
   // UNI[6435] := 16#7967;
   // UNI[6436] := 16#797A;
   // UNI[6437] := 16#7985;
   // UNI[6438] := 16#798A;
   // UNI[6439] := 16#799A;
   // UNI[6440] := 16#79A7;
   // UNI[6441] := 16#79B3;
   // UNI[6442] := 16#5FD1;
   // UNI[6443] := 16#5FD0;
   // UNI[6444] := 16#603C;
   // UNI[6445] := 16#605D;
   // UNI[6446] := 16#605A;
   // UNI[6447] := 16#6067;
   // UNI[6448] := 16#6041;
   // UNI[6449] := 16#6059;
   // UNI[6450] := 16#6063;
   // UNI[6451] := 16#60AB;
   // UNI[6452] := 16#6106;
   // UNI[6453] := 16#610D;
   // UNI[6454] := 16#615D;
   // UNI[6455] := 16#61A9;
   // UNI[6456] := 16#619D;
   // UNI[6457] := 16#61CB;
   // UNI[6458] := 16#61D1;
   // UNI[6459] := 16#6206;
   // UNI[6460] := 16#8080;
   // UNI[6461] := 16#807F;
   // UNI[6462] := 16#6C93;
   // UNI[6463] := 16#6CF6;
   // UNI[6464] := 16#6DFC;
   // UNI[6465] := 16#77F6;
   // UNI[6466] := 16#77F8;
   // UNI[6467] := 16#7800;
   // UNI[6468] := 16#7809;
   // UNI[6469] := 16#7817;
   // UNI[6470] := 16#7818;
   // UNI[6471] := 16#7811;
   // UNI[6472] := 16#65AB;
   // UNI[6473] := 16#782D;
   // UNI[6474] := 16#781C;
   // UNI[6475] := 16#781D;
   // UNI[6476] := 16#7839;
   // UNI[6477] := 16#783A;
   // UNI[6478] := 16#783B;
   // UNI[6479] := 16#781F;
   // UNI[6480] := 16#783C;
   // UNI[6481] := 16#7825;
   // UNI[6482] := 16#782C;
   // UNI[6483] := 16#7823;
   // UNI[6484] := 16#7829;
   // UNI[6485] := 16#784E;
   // UNI[6486] := 16#786D;
   // UNI[6487] := 16#7856;
   // UNI[6488] := 16#7857;
   // UNI[6489] := 16#7826;
   // UNI[6490] := 16#7850;
   // UNI[6491] := 16#7847;
   // UNI[6492] := 16#784C;
   // UNI[6493] := 16#786A;
   // UNI[6494] := 16#789B;
   // UNI[6495] := 16#7893;
   // UNI[6496] := 16#789A;
   // UNI[6497] := 16#7887;
   // UNI[6498] := 16#789C;
   // UNI[6499] := 16#78A1;
